   // GBK_TO_UNICODE[39568] := 16#F0A9;
   // GBK_TO_UNICODE[39569] := 16#7693;
   // GBK_TO_UNICODE[39570] := 16#F0AA;
   // GBK_TO_UNICODE[39571] := 16#7699;
   // GBK_TO_UNICODE[39572] := 16#F0AB;
   // GBK_TO_UNICODE[39573] := 16#76A4;
   // GBK_TO_UNICODE[39574] := 16#F0AC;
   // GBK_TO_UNICODE[39575] := 16#74DE;
   // GBK_TO_UNICODE[39576] := 16#F0AD;
   // GBK_TO_UNICODE[39577] := 16#74E0;
   // GBK_TO_UNICODE[39578] := 16#F0AE;
   // GBK_TO_UNICODE[39579] := 16#752C;
   // GBK_TO_UNICODE[39580] := 16#F0AF;
   // GBK_TO_UNICODE[39581] := 16#9E20;
   // GBK_TO_UNICODE[39582] := 16#F0B0;
   // GBK_TO_UNICODE[39583] := 16#9E22;
   // GBK_TO_UNICODE[39584] := 16#F0B1;
   // GBK_TO_UNICODE[39585] := 16#9E28;
   // GBK_TO_UNICODE[39586] := 16#F0B2;
   // GBK_TO_UNICODE[39587] := 16#9E29;
   // GBK_TO_UNICODE[39588] := 16#F0B3;
   // GBK_TO_UNICODE[39589] := 16#9E2A;
   // GBK_TO_UNICODE[39590] := 16#F0B4;
   // GBK_TO_UNICODE[39591] := 16#9E2B;
   // GBK_TO_UNICODE[39592] := 16#F0B5;
   // GBK_TO_UNICODE[39593] := 16#9E2C;
   // GBK_TO_UNICODE[39594] := 16#F0B6;
   // GBK_TO_UNICODE[39595] := 16#9E32;
   // GBK_TO_UNICODE[39596] := 16#F0B7;
   // GBK_TO_UNICODE[39597] := 16#9E31;
   // GBK_TO_UNICODE[39598] := 16#F0B8;
   // GBK_TO_UNICODE[39599] := 16#9E36;
   // GBK_TO_UNICODE[39600] := 16#F0B9;
   // GBK_TO_UNICODE[39601] := 16#9E38;
   // GBK_TO_UNICODE[39602] := 16#F0BA;
   // GBK_TO_UNICODE[39603] := 16#9E37;
   // GBK_TO_UNICODE[39604] := 16#F0BB;
   // GBK_TO_UNICODE[39605] := 16#9E39;
   // GBK_TO_UNICODE[39606] := 16#F0BC;
   // GBK_TO_UNICODE[39607] := 16#9E3A;
   // GBK_TO_UNICODE[39608] := 16#F0BD;
   // GBK_TO_UNICODE[39609] := 16#9E3E;
   // GBK_TO_UNICODE[39610] := 16#F0BE;
   // GBK_TO_UNICODE[39611] := 16#9E41;
   // GBK_TO_UNICODE[39612] := 16#F0BF;
   // GBK_TO_UNICODE[39613] := 16#9E42;
   // GBK_TO_UNICODE[39614] := 16#F0C0;
   // GBK_TO_UNICODE[39615] := 16#9E44;
   // GBK_TO_UNICODE[39616] := 16#F0C1;
   // GBK_TO_UNICODE[39617] := 16#9E46;
   // GBK_TO_UNICODE[39618] := 16#F0C2;
   // GBK_TO_UNICODE[39619] := 16#9E47;
   // GBK_TO_UNICODE[39620] := 16#F0C3;
   // GBK_TO_UNICODE[39621] := 16#9E48;
   // GBK_TO_UNICODE[39622] := 16#F0C4;
   // GBK_TO_UNICODE[39623] := 16#9E49;
   // GBK_TO_UNICODE[39624] := 16#F0C5;
   // GBK_TO_UNICODE[39625] := 16#9E4B;
   // GBK_TO_UNICODE[39626] := 16#F0C6;
   // GBK_TO_UNICODE[39627] := 16#9E4C;
   // GBK_TO_UNICODE[39628] := 16#F0C7;
   // GBK_TO_UNICODE[39629] := 16#9E4E;
   // GBK_TO_UNICODE[39630] := 16#F0C8;
   // GBK_TO_UNICODE[39631] := 16#9E51;
   // GBK_TO_UNICODE[39632] := 16#F0C9;
   // GBK_TO_UNICODE[39633] := 16#9E55;
   // GBK_TO_UNICODE[39634] := 16#F0CA;
   // GBK_TO_UNICODE[39635] := 16#9E57;
   // GBK_TO_UNICODE[39636] := 16#F0CB;
   // GBK_TO_UNICODE[39637] := 16#9E5A;
   // GBK_TO_UNICODE[39638] := 16#F0CC;
   // GBK_TO_UNICODE[39639] := 16#9E5B;
   // GBK_TO_UNICODE[39640] := 16#F0CD;
   // GBK_TO_UNICODE[39641] := 16#9E5C;
   // GBK_TO_UNICODE[39642] := 16#F0CE;
   // GBK_TO_UNICODE[39643] := 16#9E5E;
   // GBK_TO_UNICODE[39644] := 16#F0CF;
   // GBK_TO_UNICODE[39645] := 16#9E63;
   // GBK_TO_UNICODE[39646] := 16#F0D0;
   // GBK_TO_UNICODE[39647] := 16#9E66;
   // GBK_TO_UNICODE[39648] := 16#F0D1;
   // GBK_TO_UNICODE[39649] := 16#9E67;
   // GBK_TO_UNICODE[39650] := 16#F0D2;
   // GBK_TO_UNICODE[39651] := 16#9E68;
   // GBK_TO_UNICODE[39652] := 16#F0D3;
   // GBK_TO_UNICODE[39653] := 16#9E69;
   // GBK_TO_UNICODE[39654] := 16#F0D4;
   // GBK_TO_UNICODE[39655] := 16#9E6A;
   // GBK_TO_UNICODE[39656] := 16#F0D5;
   // GBK_TO_UNICODE[39657] := 16#9E6B;
   // GBK_TO_UNICODE[39658] := 16#F0D6;
   // GBK_TO_UNICODE[39659] := 16#9E6C;
   // GBK_TO_UNICODE[39660] := 16#F0D7;
   // GBK_TO_UNICODE[39661] := 16#9E71;
   // GBK_TO_UNICODE[39662] := 16#F0D8;
   // GBK_TO_UNICODE[39663] := 16#9E6D;
   // GBK_TO_UNICODE[39664] := 16#F0D9;
   // GBK_TO_UNICODE[39665] := 16#9E73;
   // GBK_TO_UNICODE[39666] := 16#F0DA;
   // GBK_TO_UNICODE[39667] := 16#7592;
   // GBK_TO_UNICODE[39668] := 16#F0DB;
   // GBK_TO_UNICODE[39669] := 16#7594;
   // GBK_TO_UNICODE[39670] := 16#F0DC;
   // GBK_TO_UNICODE[39671] := 16#7596;
   // GBK_TO_UNICODE[39672] := 16#F0DD;
   // GBK_TO_UNICODE[39673] := 16#75A0;
   // GBK_TO_UNICODE[39674] := 16#F0DE;
   // GBK_TO_UNICODE[39675] := 16#759D;
   // GBK_TO_UNICODE[39676] := 16#F0DF;
   // GBK_TO_UNICODE[39677] := 16#75AC;
   // GBK_TO_UNICODE[39678] := 16#F0E0;
   // GBK_TO_UNICODE[39679] := 16#75A3;
   // GBK_TO_UNICODE[39680] := 16#F0E1;
   // GBK_TO_UNICODE[39681] := 16#75B3;
   // GBK_TO_UNICODE[39682] := 16#F0E2;
   // GBK_TO_UNICODE[39683] := 16#75B4;
   // GBK_TO_UNICODE[39684] := 16#F0E3;
   // GBK_TO_UNICODE[39685] := 16#75B8;
   // GBK_TO_UNICODE[39686] := 16#F0E4;
   // GBK_TO_UNICODE[39687] := 16#75C4;
   // GBK_TO_UNICODE[39688] := 16#F0E5;
   // GBK_TO_UNICODE[39689] := 16#75B1;
   // GBK_TO_UNICODE[39690] := 16#F0E6;
   // GBK_TO_UNICODE[39691] := 16#75B0;
   // GBK_TO_UNICODE[39692] := 16#F0E7;
   // GBK_TO_UNICODE[39693] := 16#75C3;
   // GBK_TO_UNICODE[39694] := 16#F0E8;
   // GBK_TO_UNICODE[39695] := 16#75C2;
   // GBK_TO_UNICODE[39696] := 16#F0E9;
   // GBK_TO_UNICODE[39697] := 16#75D6;
   // GBK_TO_UNICODE[39698] := 16#F0EA;
   // GBK_TO_UNICODE[39699] := 16#75CD;
   // GBK_TO_UNICODE[39700] := 16#F0EB;
   // GBK_TO_UNICODE[39701] := 16#75E3;
   // GBK_TO_UNICODE[39702] := 16#F0EC;
   // GBK_TO_UNICODE[39703] := 16#75E8;
   // GBK_TO_UNICODE[39704] := 16#F0ED;
   // GBK_TO_UNICODE[39705] := 16#75E6;
   // GBK_TO_UNICODE[39706] := 16#F0EE;
   // GBK_TO_UNICODE[39707] := 16#75E4;
   // GBK_TO_UNICODE[39708] := 16#F0EF;
   // GBK_TO_UNICODE[39709] := 16#75EB;
   // GBK_TO_UNICODE[39710] := 16#F0F0;
   // GBK_TO_UNICODE[39711] := 16#75E7;
   // GBK_TO_UNICODE[39712] := 16#F0F1;
   // GBK_TO_UNICODE[39713] := 16#7603;
   // GBK_TO_UNICODE[39714] := 16#F0F2;
   // GBK_TO_UNICODE[39715] := 16#75F1;
   // GBK_TO_UNICODE[39716] := 16#F0F3;
   // GBK_TO_UNICODE[39717] := 16#75FC;
   // GBK_TO_UNICODE[39718] := 16#F0F4;
   // GBK_TO_UNICODE[39719] := 16#75FF;
   // GBK_TO_UNICODE[39720] := 16#F0F5;
   // GBK_TO_UNICODE[39721] := 16#7610;
   // GBK_TO_UNICODE[39722] := 16#F0F6;
   // GBK_TO_UNICODE[39723] := 16#7600;
   // GBK_TO_UNICODE[39724] := 16#F0F7;
   // GBK_TO_UNICODE[39725] := 16#7605;
   // GBK_TO_UNICODE[39726] := 16#F0F8;
   // GBK_TO_UNICODE[39727] := 16#760C;
   // GBK_TO_UNICODE[39728] := 16#F0F9;
   // GBK_TO_UNICODE[39729] := 16#7617;
   // GBK_TO_UNICODE[39730] := 16#F0FA;
   // GBK_TO_UNICODE[39731] := 16#760A;
   // GBK_TO_UNICODE[39732] := 16#F0FB;
   // GBK_TO_UNICODE[39733] := 16#7625;
   // GBK_TO_UNICODE[39734] := 16#F0FC;
   // GBK_TO_UNICODE[39735] := 16#7618;
   // GBK_TO_UNICODE[39736] := 16#F0FD;
   // GBK_TO_UNICODE[39737] := 16#7615;
   // GBK_TO_UNICODE[39738] := 16#F0FE;
   // GBK_TO_UNICODE[39739] := 16#7619;
   // GBK_TO_UNICODE[39740] := 16#F140;
   // GBK_TO_UNICODE[39741] := 16#998C;
   // GBK_TO_UNICODE[39742] := 16#F141;
   // GBK_TO_UNICODE[39743] := 16#998E;
   // GBK_TO_UNICODE[39744] := 16#F142;
   // GBK_TO_UNICODE[39745] := 16#999A;
   // GBK_TO_UNICODE[39746] := 16#F143;
   // GBK_TO_UNICODE[39747] := 16#999B;
   // GBK_TO_UNICODE[39748] := 16#F144;
   // GBK_TO_UNICODE[39749] := 16#999C;
   // GBK_TO_UNICODE[39750] := 16#F145;
   // GBK_TO_UNICODE[39751] := 16#999D;
   // GBK_TO_UNICODE[39752] := 16#F146;
   // GBK_TO_UNICODE[39753] := 16#999E;
   // GBK_TO_UNICODE[39754] := 16#F147;
   // GBK_TO_UNICODE[39755] := 16#999F;
   // GBK_TO_UNICODE[39756] := 16#F148;
   // GBK_TO_UNICODE[39757] := 16#99A0;
   // GBK_TO_UNICODE[39758] := 16#F149;
   // GBK_TO_UNICODE[39759] := 16#99A1;
   // GBK_TO_UNICODE[39760] := 16#F14A;
   // GBK_TO_UNICODE[39761] := 16#99A2;
   // GBK_TO_UNICODE[39762] := 16#F14B;
   // GBK_TO_UNICODE[39763] := 16#99A3;
   // GBK_TO_UNICODE[39764] := 16#F14C;
   // GBK_TO_UNICODE[39765] := 16#99A4;
   // GBK_TO_UNICODE[39766] := 16#F14D;
   // GBK_TO_UNICODE[39767] := 16#99A6;
   // GBK_TO_UNICODE[39768] := 16#F14E;
   // GBK_TO_UNICODE[39769] := 16#99A7;
   // GBK_TO_UNICODE[39770] := 16#F14F;
   // GBK_TO_UNICODE[39771] := 16#99A9;
   // GBK_TO_UNICODE[39772] := 16#F150;
   // GBK_TO_UNICODE[39773] := 16#99AA;
   // GBK_TO_UNICODE[39774] := 16#F151;
   // GBK_TO_UNICODE[39775] := 16#99AB;
   // GBK_TO_UNICODE[39776] := 16#F152;
   // GBK_TO_UNICODE[39777] := 16#99AC;
   // GBK_TO_UNICODE[39778] := 16#F153;
   // GBK_TO_UNICODE[39779] := 16#99AD;
   // GBK_TO_UNICODE[39780] := 16#F154;
   // GBK_TO_UNICODE[39781] := 16#99AE;
   // GBK_TO_UNICODE[39782] := 16#F155;
   // GBK_TO_UNICODE[39783] := 16#99AF;
   // GBK_TO_UNICODE[39784] := 16#F156;
   // GBK_TO_UNICODE[39785] := 16#99B0;
   // GBK_TO_UNICODE[39786] := 16#F157;
   // GBK_TO_UNICODE[39787] := 16#99B1;
   // GBK_TO_UNICODE[39788] := 16#F158;
   // GBK_TO_UNICODE[39789] := 16#99B2;
   // GBK_TO_UNICODE[39790] := 16#F159;
   // GBK_TO_UNICODE[39791] := 16#99B3;
   // GBK_TO_UNICODE[39792] := 16#F15A;
   // GBK_TO_UNICODE[39793] := 16#99B4;
   // GBK_TO_UNICODE[39794] := 16#F15B;
   // GBK_TO_UNICODE[39795] := 16#99B5;
   // GBK_TO_UNICODE[39796] := 16#F15C;
   // GBK_TO_UNICODE[39797] := 16#99B6;
   // GBK_TO_UNICODE[39798] := 16#F15D;
   // GBK_TO_UNICODE[39799] := 16#99B7;
   // GBK_TO_UNICODE[39800] := 16#F15E;
   // GBK_TO_UNICODE[39801] := 16#99B8;
   // GBK_TO_UNICODE[39802] := 16#F15F;
   // GBK_TO_UNICODE[39803] := 16#99B9;
   // GBK_TO_UNICODE[39804] := 16#F160;
   // GBK_TO_UNICODE[39805] := 16#99BA;
   // GBK_TO_UNICODE[39806] := 16#F161;
   // GBK_TO_UNICODE[39807] := 16#99BB;
   // GBK_TO_UNICODE[39808] := 16#F162;
   // GBK_TO_UNICODE[39809] := 16#99BC;
   // GBK_TO_UNICODE[39810] := 16#F163;
   // GBK_TO_UNICODE[39811] := 16#99BD;
   // GBK_TO_UNICODE[39812] := 16#F164;
   // GBK_TO_UNICODE[39813] := 16#99BE;
   // GBK_TO_UNICODE[39814] := 16#F165;
   // GBK_TO_UNICODE[39815] := 16#99BF;
   // GBK_TO_UNICODE[39816] := 16#F166;
   // GBK_TO_UNICODE[39817] := 16#99C0;
   // GBK_TO_UNICODE[39818] := 16#F167;
   // GBK_TO_UNICODE[39819] := 16#99C1;
   // GBK_TO_UNICODE[39820] := 16#F168;
   // GBK_TO_UNICODE[39821] := 16#99C2;
   // GBK_TO_UNICODE[39822] := 16#F169;
   // GBK_TO_UNICODE[39823] := 16#99C3;
   // GBK_TO_UNICODE[39824] := 16#F16A;
   // GBK_TO_UNICODE[39825] := 16#99C4;
   // GBK_TO_UNICODE[39826] := 16#F16B;
   // GBK_TO_UNICODE[39827] := 16#99C5;
   // GBK_TO_UNICODE[39828] := 16#F16C;
   // GBK_TO_UNICODE[39829] := 16#99C6;
   // GBK_TO_UNICODE[39830] := 16#F16D;
   // GBK_TO_UNICODE[39831] := 16#99C7;
   // GBK_TO_UNICODE[39832] := 16#F16E;
   // GBK_TO_UNICODE[39833] := 16#99C8;
   // GBK_TO_UNICODE[39834] := 16#F16F;
   // GBK_TO_UNICODE[39835] := 16#99C9;
   // GBK_TO_UNICODE[39836] := 16#F170;
   // GBK_TO_UNICODE[39837] := 16#99CA;
   // GBK_TO_UNICODE[39838] := 16#F171;
   // GBK_TO_UNICODE[39839] := 16#99CB;
   // GBK_TO_UNICODE[39840] := 16#F172;
   // GBK_TO_UNICODE[39841] := 16#99CC;
   // GBK_TO_UNICODE[39842] := 16#F173;
   // GBK_TO_UNICODE[39843] := 16#99CD;
   // GBK_TO_UNICODE[39844] := 16#F174;
   // GBK_TO_UNICODE[39845] := 16#99CE;
   // GBK_TO_UNICODE[39846] := 16#F175;
   // GBK_TO_UNICODE[39847] := 16#99CF;
   // GBK_TO_UNICODE[39848] := 16#F176;
   // GBK_TO_UNICODE[39849] := 16#99D0;
   // GBK_TO_UNICODE[39850] := 16#F177;
   // GBK_TO_UNICODE[39851] := 16#99D1;
   // GBK_TO_UNICODE[39852] := 16#F178;
   // GBK_TO_UNICODE[39853] := 16#99D2;
   // GBK_TO_UNICODE[39854] := 16#F179;
   // GBK_TO_UNICODE[39855] := 16#99D3;
   // GBK_TO_UNICODE[39856] := 16#F17A;
   // GBK_TO_UNICODE[39857] := 16#99D4;
   // GBK_TO_UNICODE[39858] := 16#F17B;
   // GBK_TO_UNICODE[39859] := 16#99D5;
   // GBK_TO_UNICODE[39860] := 16#F17C;
   // GBK_TO_UNICODE[39861] := 16#99D6;
   // GBK_TO_UNICODE[39862] := 16#F17D;
   // GBK_TO_UNICODE[39863] := 16#99D7;
   // GBK_TO_UNICODE[39864] := 16#F17E;
   // GBK_TO_UNICODE[39865] := 16#99D8;
   // GBK_TO_UNICODE[39866] := 16#F180;
   // GBK_TO_UNICODE[39867] := 16#99D9;
   // GBK_TO_UNICODE[39868] := 16#F181;
   // GBK_TO_UNICODE[39869] := 16#99DA;
   // GBK_TO_UNICODE[39870] := 16#F182;
   // GBK_TO_UNICODE[39871] := 16#99DB;
   // GBK_TO_UNICODE[39872] := 16#F183;
   // GBK_TO_UNICODE[39873] := 16#99DC;
   // GBK_TO_UNICODE[39874] := 16#F184;
   // GBK_TO_UNICODE[39875] := 16#99DD;
   // GBK_TO_UNICODE[39876] := 16#F185;
   // GBK_TO_UNICODE[39877] := 16#99DE;
   // GBK_TO_UNICODE[39878] := 16#F186;
   // GBK_TO_UNICODE[39879] := 16#99DF;
   // GBK_TO_UNICODE[39880] := 16#F187;
   // GBK_TO_UNICODE[39881] := 16#99E0;
   // GBK_TO_UNICODE[39882] := 16#F188;
   // GBK_TO_UNICODE[39883] := 16#99E1;
   // GBK_TO_UNICODE[39884] := 16#F189;
   // GBK_TO_UNICODE[39885] := 16#99E2;
   // GBK_TO_UNICODE[39886] := 16#F18A;
   // GBK_TO_UNICODE[39887] := 16#99E3;
   // GBK_TO_UNICODE[39888] := 16#F18B;
   // GBK_TO_UNICODE[39889] := 16#99E4;
   // GBK_TO_UNICODE[39890] := 16#F18C;
   // GBK_TO_UNICODE[39891] := 16#99E5;
   // GBK_TO_UNICODE[39892] := 16#F18D;
   // GBK_TO_UNICODE[39893] := 16#99E6;
   // GBK_TO_UNICODE[39894] := 16#F18E;
   // GBK_TO_UNICODE[39895] := 16#99E7;
   // GBK_TO_UNICODE[39896] := 16#F18F;
   // GBK_TO_UNICODE[39897] := 16#99E8;
   // GBK_TO_UNICODE[39898] := 16#F190;
   // GBK_TO_UNICODE[39899] := 16#99E9;
   // GBK_TO_UNICODE[39900] := 16#F191;
   // GBK_TO_UNICODE[39901] := 16#99EA;
   // GBK_TO_UNICODE[39902] := 16#F192;
   // GBK_TO_UNICODE[39903] := 16#99EB;
   // GBK_TO_UNICODE[39904] := 16#F193;
   // GBK_TO_UNICODE[39905] := 16#99EC;
   // GBK_TO_UNICODE[39906] := 16#F194;
   // GBK_TO_UNICODE[39907] := 16#99ED;
   // GBK_TO_UNICODE[39908] := 16#F195;
   // GBK_TO_UNICODE[39909] := 16#99EE;
   // GBK_TO_UNICODE[39910] := 16#F196;
   // GBK_TO_UNICODE[39911] := 16#99EF;
   // GBK_TO_UNICODE[39912] := 16#F197;
   // GBK_TO_UNICODE[39913] := 16#99F0;
   // GBK_TO_UNICODE[39914] := 16#F198;
   // GBK_TO_UNICODE[39915] := 16#99F1;
   // GBK_TO_UNICODE[39916] := 16#F199;
   // GBK_TO_UNICODE[39917] := 16#99F2;
   // GBK_TO_UNICODE[39918] := 16#F19A;
   // GBK_TO_UNICODE[39919] := 16#99F3;
   // GBK_TO_UNICODE[39920] := 16#F19B;
   // GBK_TO_UNICODE[39921] := 16#99F4;
   // GBK_TO_UNICODE[39922] := 16#F19C;
   // GBK_TO_UNICODE[39923] := 16#99F5;
   // GBK_TO_UNICODE[39924] := 16#F19D;
   // GBK_TO_UNICODE[39925] := 16#99F6;
   // GBK_TO_UNICODE[39926] := 16#F19E;
   // GBK_TO_UNICODE[39927] := 16#99F7;
   // GBK_TO_UNICODE[39928] := 16#F19F;
   // GBK_TO_UNICODE[39929] := 16#99F8;
   // GBK_TO_UNICODE[39930] := 16#F1A0;
   // GBK_TO_UNICODE[39931] := 16#99F9;
   // GBK_TO_UNICODE[39932] := 16#F1A1;
   // GBK_TO_UNICODE[39933] := 16#761B;
   // GBK_TO_UNICODE[39934] := 16#F1A2;
   // GBK_TO_UNICODE[39935] := 16#763C;
   // GBK_TO_UNICODE[39936] := 16#F1A3;
   // GBK_TO_UNICODE[39937] := 16#7622;
   // GBK_TO_UNICODE[39938] := 16#F1A4;
   // GBK_TO_UNICODE[39939] := 16#7620;
   // GBK_TO_UNICODE[39940] := 16#F1A5;
   // GBK_TO_UNICODE[39941] := 16#7640;
   // GBK_TO_UNICODE[39942] := 16#F1A6;
   // GBK_TO_UNICODE[39943] := 16#762D;
   // GBK_TO_UNICODE[39944] := 16#F1A7;
   // GBK_TO_UNICODE[39945] := 16#7630;
   // GBK_TO_UNICODE[39946] := 16#F1A8;
   // GBK_TO_UNICODE[39947] := 16#763F;
   // GBK_TO_UNICODE[39948] := 16#F1A9;
   // GBK_TO_UNICODE[39949] := 16#7635;
   // GBK_TO_UNICODE[39950] := 16#F1AA;
   // GBK_TO_UNICODE[39951] := 16#7643;
   // GBK_TO_UNICODE[39952] := 16#F1AB;
   // GBK_TO_UNICODE[39953] := 16#763E;
   // GBK_TO_UNICODE[39954] := 16#F1AC;
   // GBK_TO_UNICODE[39955] := 16#7633;
   // GBK_TO_UNICODE[39956] := 16#F1AD;
   // GBK_TO_UNICODE[39957] := 16#764D;
   // GBK_TO_UNICODE[39958] := 16#F1AE;
   // GBK_TO_UNICODE[39959] := 16#765E;
   // GBK_TO_UNICODE[39960] := 16#F1AF;
   // GBK_TO_UNICODE[39961] := 16#7654;
   // GBK_TO_UNICODE[39962] := 16#F1B0;
   // GBK_TO_UNICODE[39963] := 16#765C;
   // GBK_TO_UNICODE[39964] := 16#F1B1;
   // GBK_TO_UNICODE[39965] := 16#7656;
   // GBK_TO_UNICODE[39966] := 16#F1B2;
   // GBK_TO_UNICODE[39967] := 16#766B;
   // GBK_TO_UNICODE[39968] := 16#F1B3;
   // GBK_TO_UNICODE[39969] := 16#766F;
   // GBK_TO_UNICODE[39970] := 16#F1B4;
   // GBK_TO_UNICODE[39971] := 16#7FCA;
   // GBK_TO_UNICODE[39972] := 16#F1B5;
   // GBK_TO_UNICODE[39973] := 16#7AE6;
   // GBK_TO_UNICODE[39974] := 16#F1B6;
   // GBK_TO_UNICODE[39975] := 16#7A78;
   // GBK_TO_UNICODE[39976] := 16#F1B7;
   // GBK_TO_UNICODE[39977] := 16#7A79;
   // GBK_TO_UNICODE[39978] := 16#F1B8;
   // GBK_TO_UNICODE[39979] := 16#7A80;
   // GBK_TO_UNICODE[39980] := 16#F1B9;
   // GBK_TO_UNICODE[39981] := 16#7A86;
   // GBK_TO_UNICODE[39982] := 16#F1BA;
   // GBK_TO_UNICODE[39983] := 16#7A88;
   // GBK_TO_UNICODE[39984] := 16#F1BB;
   // GBK_TO_UNICODE[39985] := 16#7A95;
   // GBK_TO_UNICODE[39986] := 16#F1BC;
   // GBK_TO_UNICODE[39987] := 16#7AA6;
   // GBK_TO_UNICODE[39988] := 16#F1BD;
   // GBK_TO_UNICODE[39989] := 16#7AA0;
   // GBK_TO_UNICODE[39990] := 16#F1BE;
   // GBK_TO_UNICODE[39991] := 16#7AAC;
   // GBK_TO_UNICODE[39992] := 16#F1BF;
   // GBK_TO_UNICODE[39993] := 16#7AA8;
   // GBK_TO_UNICODE[39994] := 16#F1C0;
   // GBK_TO_UNICODE[39995] := 16#7AAD;
   // GBK_TO_UNICODE[39996] := 16#F1C1;
   // GBK_TO_UNICODE[39997] := 16#7AB3;
   // GBK_TO_UNICODE[39998] := 16#F1C2;
   // GBK_TO_UNICODE[39999] := 16#8864;
   // GBK_TO_UNICODE[40000] := 16#F1C3;
   // GBK_TO_UNICODE[40001] := 16#8869;
   // GBK_TO_UNICODE[40002] := 16#F1C4;
   // GBK_TO_UNICODE[40003] := 16#8872;
   // GBK_TO_UNICODE[40004] := 16#F1C5;
   // GBK_TO_UNICODE[40005] := 16#887D;
   // GBK_TO_UNICODE[40006] := 16#F1C6;
   // GBK_TO_UNICODE[40007] := 16#887F;
   // GBK_TO_UNICODE[40008] := 16#F1C7;
   // GBK_TO_UNICODE[40009] := 16#8882;
   // GBK_TO_UNICODE[40010] := 16#F1C8;
   // GBK_TO_UNICODE[40011] := 16#88A2;
   // GBK_TO_UNICODE[40012] := 16#F1C9;
   // GBK_TO_UNICODE[40013] := 16#88C6;
   // GBK_TO_UNICODE[40014] := 16#F1CA;
   // GBK_TO_UNICODE[40015] := 16#88B7;
   // GBK_TO_UNICODE[40016] := 16#F1CB;
   // GBK_TO_UNICODE[40017] := 16#88BC;
   // GBK_TO_UNICODE[40018] := 16#F1CC;
   // GBK_TO_UNICODE[40019] := 16#88C9;
   // GBK_TO_UNICODE[40020] := 16#F1CD;
   // GBK_TO_UNICODE[40021] := 16#88E2;
   // GBK_TO_UNICODE[40022] := 16#F1CE;
   // GBK_TO_UNICODE[40023] := 16#88CE;
   // GBK_TO_UNICODE[40024] := 16#F1CF;
   // GBK_TO_UNICODE[40025] := 16#88E3;
   // GBK_TO_UNICODE[40026] := 16#F1D0;
   // GBK_TO_UNICODE[40027] := 16#88E5;
   // GBK_TO_UNICODE[40028] := 16#F1D1;
   // GBK_TO_UNICODE[40029] := 16#88F1;
   // GBK_TO_UNICODE[40030] := 16#F1D2;
   // GBK_TO_UNICODE[40031] := 16#891A;
   // GBK_TO_UNICODE[40032] := 16#F1D3;
   // GBK_TO_UNICODE[40033] := 16#88FC;
   // GBK_TO_UNICODE[40034] := 16#F1D4;
   // GBK_TO_UNICODE[40035] := 16#88E8;
   // GBK_TO_UNICODE[40036] := 16#F1D5;
   // GBK_TO_UNICODE[40037] := 16#88FE;
   // GBK_TO_UNICODE[40038] := 16#F1D6;
   // GBK_TO_UNICODE[40039] := 16#88F0;
   // GBK_TO_UNICODE[40040] := 16#F1D7;
   // GBK_TO_UNICODE[40041] := 16#8921;
   // GBK_TO_UNICODE[40042] := 16#F1D8;
   // GBK_TO_UNICODE[40043] := 16#8919;
   // GBK_TO_UNICODE[40044] := 16#F1D9;
   // GBK_TO_UNICODE[40045] := 16#8913;
   // GBK_TO_UNICODE[40046] := 16#F1DA;
   // GBK_TO_UNICODE[40047] := 16#891B;
   // GBK_TO_UNICODE[40048] := 16#F1DB;
   // GBK_TO_UNICODE[40049] := 16#890A;
   // GBK_TO_UNICODE[40050] := 16#F1DC;
   // GBK_TO_UNICODE[40051] := 16#8934;
   // GBK_TO_UNICODE[40052] := 16#F1DD;
   // GBK_TO_UNICODE[40053] := 16#892B;
   // GBK_TO_UNICODE[40054] := 16#F1DE;
   // GBK_TO_UNICODE[40055] := 16#8936;
   // GBK_TO_UNICODE[40056] := 16#F1DF;
   // GBK_TO_UNICODE[40057] := 16#8941;
   // GBK_TO_UNICODE[40058] := 16#F1E0;
   // GBK_TO_UNICODE[40059] := 16#8966;
   // GBK_TO_UNICODE[40060] := 16#F1E1;
   // GBK_TO_UNICODE[40061] := 16#897B;
   // GBK_TO_UNICODE[40062] := 16#F1E2;
   // GBK_TO_UNICODE[40063] := 16#758B;
   // GBK_TO_UNICODE[40064] := 16#F1E3;
   // GBK_TO_UNICODE[40065] := 16#80E5;
   // GBK_TO_UNICODE[40066] := 16#F1E4;
   // GBK_TO_UNICODE[40067] := 16#76B2;
   // GBK_TO_UNICODE[40068] := 16#F1E5;
   // GBK_TO_UNICODE[40069] := 16#76B4;
   // GBK_TO_UNICODE[40070] := 16#F1E6;
   // GBK_TO_UNICODE[40071] := 16#77DC;
   // GBK_TO_UNICODE[40072] := 16#F1E7;
   // GBK_TO_UNICODE[40073] := 16#8012;
   // GBK_TO_UNICODE[40074] := 16#F1E8;
   // GBK_TO_UNICODE[40075] := 16#8014;
   // GBK_TO_UNICODE[40076] := 16#F1E9;
   // GBK_TO_UNICODE[40077] := 16#8016;
   // GBK_TO_UNICODE[40078] := 16#F1EA;
   // GBK_TO_UNICODE[40079] := 16#801C;
   // GBK_TO_UNICODE[40080] := 16#F1EB;
   // GBK_TO_UNICODE[40081] := 16#8020;
   // GBK_TO_UNICODE[40082] := 16#F1EC;
   // GBK_TO_UNICODE[40083] := 16#8022;
   // GBK_TO_UNICODE[40084] := 16#F1ED;
   // GBK_TO_UNICODE[40085] := 16#8025;
   // GBK_TO_UNICODE[40086] := 16#F1EE;
   // GBK_TO_UNICODE[40087] := 16#8026;
   // GBK_TO_UNICODE[40088] := 16#F1EF;
   // GBK_TO_UNICODE[40089] := 16#8027;
   // GBK_TO_UNICODE[40090] := 16#F1F0;
   // GBK_TO_UNICODE[40091] := 16#8029;
   // GBK_TO_UNICODE[40092] := 16#F1F1;
   // GBK_TO_UNICODE[40093] := 16#8028;
   // GBK_TO_UNICODE[40094] := 16#F1F2;
   // GBK_TO_UNICODE[40095] := 16#8031;
   // GBK_TO_UNICODE[40096] := 16#F1F3;
   // GBK_TO_UNICODE[40097] := 16#800B;
   // GBK_TO_UNICODE[40098] := 16#F1F4;
   // GBK_TO_UNICODE[40099] := 16#8035;
   // GBK_TO_UNICODE[40100] := 16#F1F5;
   // GBK_TO_UNICODE[40101] := 16#8043;
   // GBK_TO_UNICODE[40102] := 16#F1F6;
   // GBK_TO_UNICODE[40103] := 16#8046;
   // GBK_TO_UNICODE[40104] := 16#F1F7;
   // GBK_TO_UNICODE[40105] := 16#804D;
   // GBK_TO_UNICODE[40106] := 16#F1F8;
   // GBK_TO_UNICODE[40107] := 16#8052;
   // GBK_TO_UNICODE[40108] := 16#F1F9;
   // GBK_TO_UNICODE[40109] := 16#8069;
   // GBK_TO_UNICODE[40110] := 16#F1FA;
   // GBK_TO_UNICODE[40111] := 16#8071;
   // GBK_TO_UNICODE[40112] := 16#F1FB;
   // GBK_TO_UNICODE[40113] := 16#8983;
   // GBK_TO_UNICODE[40114] := 16#F1FC;
   // GBK_TO_UNICODE[40115] := 16#9878;
   // GBK_TO_UNICODE[40116] := 16#F1FD;
   // GBK_TO_UNICODE[40117] := 16#9880;
   // GBK_TO_UNICODE[40118] := 16#F1FE;
   // GBK_TO_UNICODE[40119] := 16#9883;
   // GBK_TO_UNICODE[40120] := 16#F240;
   // GBK_TO_UNICODE[40121] := 16#99FA;
   // GBK_TO_UNICODE[40122] := 16#F241;
   // GBK_TO_UNICODE[40123] := 16#99FB;
   // GBK_TO_UNICODE[40124] := 16#F242;
   // GBK_TO_UNICODE[40125] := 16#99FC;
   // GBK_TO_UNICODE[40126] := 16#F243;
   // GBK_TO_UNICODE[40127] := 16#99FD;
   // GBK_TO_UNICODE[40128] := 16#F244;
   // GBK_TO_UNICODE[40129] := 16#99FE;
   // GBK_TO_UNICODE[40130] := 16#F245;
   // GBK_TO_UNICODE[40131] := 16#99FF;
   // GBK_TO_UNICODE[40132] := 16#F246;
   // GBK_TO_UNICODE[40133] := 16#9A00;
   // GBK_TO_UNICODE[40134] := 16#F247;
   // GBK_TO_UNICODE[40135] := 16#9A01;
   // GBK_TO_UNICODE[40136] := 16#F248;
   // GBK_TO_UNICODE[40137] := 16#9A02;
   // GBK_TO_UNICODE[40138] := 16#F249;
   // GBK_TO_UNICODE[40139] := 16#9A03;
   // GBK_TO_UNICODE[40140] := 16#F24A;
   // GBK_TO_UNICODE[40141] := 16#9A04;
   // GBK_TO_UNICODE[40142] := 16#F24B;
   // GBK_TO_UNICODE[40143] := 16#9A05;
   // GBK_TO_UNICODE[40144] := 16#F24C;
   // GBK_TO_UNICODE[40145] := 16#9A06;
   // GBK_TO_UNICODE[40146] := 16#F24D;
   // GBK_TO_UNICODE[40147] := 16#9A07;
   // GBK_TO_UNICODE[40148] := 16#F24E;
   // GBK_TO_UNICODE[40149] := 16#9A08;
   // GBK_TO_UNICODE[40150] := 16#F24F;
   // GBK_TO_UNICODE[40151] := 16#9A09;
   // GBK_TO_UNICODE[40152] := 16#F250;
   // GBK_TO_UNICODE[40153] := 16#9A0A;
   // GBK_TO_UNICODE[40154] := 16#F251;
   // GBK_TO_UNICODE[40155] := 16#9A0B;
   // GBK_TO_UNICODE[40156] := 16#F252;
   // GBK_TO_UNICODE[40157] := 16#9A0C;
   // GBK_TO_UNICODE[40158] := 16#F253;
   // GBK_TO_UNICODE[40159] := 16#9A0D;
   // GBK_TO_UNICODE[40160] := 16#F254;
   // GBK_TO_UNICODE[40161] := 16#9A0E;
   // GBK_TO_UNICODE[40162] := 16#F255;
   // GBK_TO_UNICODE[40163] := 16#9A0F;
   // GBK_TO_UNICODE[40164] := 16#F256;
   // GBK_TO_UNICODE[40165] := 16#9A10;
   // GBK_TO_UNICODE[40166] := 16#F257;
   // GBK_TO_UNICODE[40167] := 16#9A11;
   // GBK_TO_UNICODE[40168] := 16#F258;
   // GBK_TO_UNICODE[40169] := 16#9A12;
   // GBK_TO_UNICODE[40170] := 16#F259;
   // GBK_TO_UNICODE[40171] := 16#9A13;
   // GBK_TO_UNICODE[40172] := 16#F25A;
   // GBK_TO_UNICODE[40173] := 16#9A14;
   // GBK_TO_UNICODE[40174] := 16#F25B;
   // GBK_TO_UNICODE[40175] := 16#9A15;
   // GBK_TO_UNICODE[40176] := 16#F25C;
   // GBK_TO_UNICODE[40177] := 16#9A16;
   // GBK_TO_UNICODE[40178] := 16#F25D;
   // GBK_TO_UNICODE[40179] := 16#9A17;
   // GBK_TO_UNICODE[40180] := 16#F25E;
   // GBK_TO_UNICODE[40181] := 16#9A18;
   // GBK_TO_UNICODE[40182] := 16#F25F;
   // GBK_TO_UNICODE[40183] := 16#9A19;
   // GBK_TO_UNICODE[40184] := 16#F260;
   // GBK_TO_UNICODE[40185] := 16#9A1A;
   // GBK_TO_UNICODE[40186] := 16#F261;
   // GBK_TO_UNICODE[40187] := 16#9A1B;
   // GBK_TO_UNICODE[40188] := 16#F262;
   // GBK_TO_UNICODE[40189] := 16#9A1C;
   // GBK_TO_UNICODE[40190] := 16#F263;
   // GBK_TO_UNICODE[40191] := 16#9A1D;
   // GBK_TO_UNICODE[40192] := 16#F264;
   // GBK_TO_UNICODE[40193] := 16#9A1E;
   // GBK_TO_UNICODE[40194] := 16#F265;
   // GBK_TO_UNICODE[40195] := 16#9A1F;
   // GBK_TO_UNICODE[40196] := 16#F266;
   // GBK_TO_UNICODE[40197] := 16#9A20;
   // GBK_TO_UNICODE[40198] := 16#F267;
   // GBK_TO_UNICODE[40199] := 16#9A21;
   // GBK_TO_UNICODE[40200] := 16#F268;
   // GBK_TO_UNICODE[40201] := 16#9A22;
   // GBK_TO_UNICODE[40202] := 16#F269;
   // GBK_TO_UNICODE[40203] := 16#9A23;
   // GBK_TO_UNICODE[40204] := 16#F26A;
   // GBK_TO_UNICODE[40205] := 16#9A24;
   // GBK_TO_UNICODE[40206] := 16#F26B;
   // GBK_TO_UNICODE[40207] := 16#9A25;
   // GBK_TO_UNICODE[40208] := 16#F26C;
   // GBK_TO_UNICODE[40209] := 16#9A26;
   // GBK_TO_UNICODE[40210] := 16#F26D;
   // GBK_TO_UNICODE[40211] := 16#9A27;
   // GBK_TO_UNICODE[40212] := 16#F26E;
   // GBK_TO_UNICODE[40213] := 16#9A28;
   // GBK_TO_UNICODE[40214] := 16#F26F;
   // GBK_TO_UNICODE[40215] := 16#9A29;
   // GBK_TO_UNICODE[40216] := 16#F270;
   // GBK_TO_UNICODE[40217] := 16#9A2A;
   // GBK_TO_UNICODE[40218] := 16#F271;
   // GBK_TO_UNICODE[40219] := 16#9A2B;
   // GBK_TO_UNICODE[40220] := 16#F272;
   // GBK_TO_UNICODE[40221] := 16#9A2C;
   // GBK_TO_UNICODE[40222] := 16#F273;
   // GBK_TO_UNICODE[40223] := 16#9A2D;
   // GBK_TO_UNICODE[40224] := 16#F274;
   // GBK_TO_UNICODE[40225] := 16#9A2E;
   // GBK_TO_UNICODE[40226] := 16#F275;
   // GBK_TO_UNICODE[40227] := 16#9A2F;
   // GBK_TO_UNICODE[40228] := 16#F276;
   // GBK_TO_UNICODE[40229] := 16#9A30;
   // GBK_TO_UNICODE[40230] := 16#F277;
   // GBK_TO_UNICODE[40231] := 16#9A31;
   // GBK_TO_UNICODE[40232] := 16#F278;
   // GBK_TO_UNICODE[40233] := 16#9A32;
   // GBK_TO_UNICODE[40234] := 16#F279;
   // GBK_TO_UNICODE[40235] := 16#9A33;
   // GBK_TO_UNICODE[40236] := 16#F27A;
   // GBK_TO_UNICODE[40237] := 16#9A34;
   // GBK_TO_UNICODE[40238] := 16#F27B;
   // GBK_TO_UNICODE[40239] := 16#9A35;
   // GBK_TO_UNICODE[40240] := 16#F27C;
   // GBK_TO_UNICODE[40241] := 16#9A36;
   // GBK_TO_UNICODE[40242] := 16#F27D;
   // GBK_TO_UNICODE[40243] := 16#9A37;
   // GBK_TO_UNICODE[40244] := 16#F27E;
   // GBK_TO_UNICODE[40245] := 16#9A38;
   // GBK_TO_UNICODE[40246] := 16#F280;
   // GBK_TO_UNICODE[40247] := 16#9A39;
   // GBK_TO_UNICODE[40248] := 16#F281;
   // GBK_TO_UNICODE[40249] := 16#9A3A;
   // GBK_TO_UNICODE[40250] := 16#F282;
   // GBK_TO_UNICODE[40251] := 16#9A3B;
   // GBK_TO_UNICODE[40252] := 16#F283;
   // GBK_TO_UNICODE[40253] := 16#9A3C;
   // GBK_TO_UNICODE[40254] := 16#F284;
   // GBK_TO_UNICODE[40255] := 16#9A3D;
   // GBK_TO_UNICODE[40256] := 16#F285;
   // GBK_TO_UNICODE[40257] := 16#9A3E;
   // GBK_TO_UNICODE[40258] := 16#F286;
   // GBK_TO_UNICODE[40259] := 16#9A3F;
   // GBK_TO_UNICODE[40260] := 16#F287;
   // GBK_TO_UNICODE[40261] := 16#9A40;
   // GBK_TO_UNICODE[40262] := 16#F288;
   // GBK_TO_UNICODE[40263] := 16#9A41;
   // GBK_TO_UNICODE[40264] := 16#F289;
   // GBK_TO_UNICODE[40265] := 16#9A42;
   // GBK_TO_UNICODE[40266] := 16#F28A;
   // GBK_TO_UNICODE[40267] := 16#9A43;
   // GBK_TO_UNICODE[40268] := 16#F28B;
   // GBK_TO_UNICODE[40269] := 16#9A44;
   // GBK_TO_UNICODE[40270] := 16#F28C;
   // GBK_TO_UNICODE[40271] := 16#9A45;
   // GBK_TO_UNICODE[40272] := 16#F28D;
   // GBK_TO_UNICODE[40273] := 16#9A46;
   // GBK_TO_UNICODE[40274] := 16#F28E;
   // GBK_TO_UNICODE[40275] := 16#9A47;
   // GBK_TO_UNICODE[40276] := 16#F28F;
   // GBK_TO_UNICODE[40277] := 16#9A48;
   // GBK_TO_UNICODE[40278] := 16#F290;
   // GBK_TO_UNICODE[40279] := 16#9A49;
   // GBK_TO_UNICODE[40280] := 16#F291;
   // GBK_TO_UNICODE[40281] := 16#9A4A;
   // GBK_TO_UNICODE[40282] := 16#F292;
   // GBK_TO_UNICODE[40283] := 16#9A4B;
   // GBK_TO_UNICODE[40284] := 16#F293;
   // GBK_TO_UNICODE[40285] := 16#9A4C;
   // GBK_TO_UNICODE[40286] := 16#F294;
   // GBK_TO_UNICODE[40287] := 16#9A4D;
   // GBK_TO_UNICODE[40288] := 16#F295;
   // GBK_TO_UNICODE[40289] := 16#9A4E;
   // GBK_TO_UNICODE[40290] := 16#F296;
   // GBK_TO_UNICODE[40291] := 16#9A4F;
   // GBK_TO_UNICODE[40292] := 16#F297;
   // GBK_TO_UNICODE[40293] := 16#9A50;
   // GBK_TO_UNICODE[40294] := 16#F298;
   // GBK_TO_UNICODE[40295] := 16#9A51;
   // GBK_TO_UNICODE[40296] := 16#F299;
   // GBK_TO_UNICODE[40297] := 16#9A52;
   // GBK_TO_UNICODE[40298] := 16#F29A;
   // GBK_TO_UNICODE[40299] := 16#9A53;
   // GBK_TO_UNICODE[40300] := 16#F29B;
   // GBK_TO_UNICODE[40301] := 16#9A54;
   // GBK_TO_UNICODE[40302] := 16#F29C;
   // GBK_TO_UNICODE[40303] := 16#9A55;
   // GBK_TO_UNICODE[40304] := 16#F29D;
   // GBK_TO_UNICODE[40305] := 16#9A56;
   // GBK_TO_UNICODE[40306] := 16#F29E;
   // GBK_TO_UNICODE[40307] := 16#9A57;
   // GBK_TO_UNICODE[40308] := 16#F29F;
   // GBK_TO_UNICODE[40309] := 16#9A58;
   // GBK_TO_UNICODE[40310] := 16#F2A0;
   // GBK_TO_UNICODE[40311] := 16#9A59;
   // GBK_TO_UNICODE[40312] := 16#F2A1;
   // GBK_TO_UNICODE[40313] := 16#9889;
   // GBK_TO_UNICODE[40314] := 16#F2A2;
   // GBK_TO_UNICODE[40315] := 16#988C;
   // GBK_TO_UNICODE[40316] := 16#F2A3;
   // GBK_TO_UNICODE[40317] := 16#988D;
   // GBK_TO_UNICODE[40318] := 16#F2A4;
   // GBK_TO_UNICODE[40319] := 16#988F;
   // GBK_TO_UNICODE[40320] := 16#F2A5;
   // GBK_TO_UNICODE[40321] := 16#9894;
   // GBK_TO_UNICODE[40322] := 16#F2A6;
   // GBK_TO_UNICODE[40323] := 16#989A;
   // GBK_TO_UNICODE[40324] := 16#F2A7;
   // GBK_TO_UNICODE[40325] := 16#989B;
   // GBK_TO_UNICODE[40326] := 16#F2A8;
   // GBK_TO_UNICODE[40327] := 16#989E;
   // GBK_TO_UNICODE[40328] := 16#F2A9;
   // GBK_TO_UNICODE[40329] := 16#989F;
   // GBK_TO_UNICODE[40330] := 16#F2AA;
   // GBK_TO_UNICODE[40331] := 16#98A1;
   // GBK_TO_UNICODE[40332] := 16#F2AB;
   // GBK_TO_UNICODE[40333] := 16#98A2;
   // GBK_TO_UNICODE[40334] := 16#F2AC;
   // GBK_TO_UNICODE[40335] := 16#98A5;
   // GBK_TO_UNICODE[40336] := 16#F2AD;
   // GBK_TO_UNICODE[40337] := 16#98A6;
   // GBK_TO_UNICODE[40338] := 16#F2AE;
   // GBK_TO_UNICODE[40339] := 16#864D;
   // GBK_TO_UNICODE[40340] := 16#F2AF;
   // GBK_TO_UNICODE[40341] := 16#8654;
   // GBK_TO_UNICODE[40342] := 16#F2B0;
   // GBK_TO_UNICODE[40343] := 16#866C;
   // GBK_TO_UNICODE[40344] := 16#F2B1;
   // GBK_TO_UNICODE[40345] := 16#866E;
   // GBK_TO_UNICODE[40346] := 16#F2B2;
   // GBK_TO_UNICODE[40347] := 16#867F;
   // GBK_TO_UNICODE[40348] := 16#F2B3;
   // GBK_TO_UNICODE[40349] := 16#867A;
   // GBK_TO_UNICODE[40350] := 16#F2B4;
   // GBK_TO_UNICODE[40351] := 16#867C;
   // GBK_TO_UNICODE[40352] := 16#F2B5;
   // GBK_TO_UNICODE[40353] := 16#867B;
   // GBK_TO_UNICODE[40354] := 16#F2B6;
   // GBK_TO_UNICODE[40355] := 16#86A8;
   // GBK_TO_UNICODE[40356] := 16#F2B7;
   // GBK_TO_UNICODE[40357] := 16#868D;
   // GBK_TO_UNICODE[40358] := 16#F2B8;
   // GBK_TO_UNICODE[40359] := 16#868B;
   // GBK_TO_UNICODE[40360] := 16#F2B9;
   // GBK_TO_UNICODE[40361] := 16#86AC;
   // GBK_TO_UNICODE[40362] := 16#F2BA;
   // GBK_TO_UNICODE[40363] := 16#869D;
   // GBK_TO_UNICODE[40364] := 16#F2BB;
   // GBK_TO_UNICODE[40365] := 16#86A7;
   // GBK_TO_UNICODE[40366] := 16#F2BC;
   // GBK_TO_UNICODE[40367] := 16#86A3;
   // GBK_TO_UNICODE[40368] := 16#F2BD;
   // GBK_TO_UNICODE[40369] := 16#86AA;
   // GBK_TO_UNICODE[40370] := 16#F2BE;
   // GBK_TO_UNICODE[40371] := 16#8693;
   // GBK_TO_UNICODE[40372] := 16#F2BF;
   // GBK_TO_UNICODE[40373] := 16#86A9;
   // GBK_TO_UNICODE[40374] := 16#F2C0;
   // GBK_TO_UNICODE[40375] := 16#86B6;
   // GBK_TO_UNICODE[40376] := 16#F2C1;
   // GBK_TO_UNICODE[40377] := 16#86C4;
   // GBK_TO_UNICODE[40378] := 16#F2C2;
   // GBK_TO_UNICODE[40379] := 16#86B5;
   // GBK_TO_UNICODE[40380] := 16#F2C3;
   // GBK_TO_UNICODE[40381] := 16#86CE;
   // GBK_TO_UNICODE[40382] := 16#F2C4;
   // GBK_TO_UNICODE[40383] := 16#86B0;
   // GBK_TO_UNICODE[40384] := 16#F2C5;
   // GBK_TO_UNICODE[40385] := 16#86BA;
   // GBK_TO_UNICODE[40386] := 16#F2C6;
   // GBK_TO_UNICODE[40387] := 16#86B1;
   // GBK_TO_UNICODE[40388] := 16#F2C7;
   // GBK_TO_UNICODE[40389] := 16#86AF;
   // GBK_TO_UNICODE[40390] := 16#F2C8;
   // GBK_TO_UNICODE[40391] := 16#86C9;
   // GBK_TO_UNICODE[40392] := 16#F2C9;
   // GBK_TO_UNICODE[40393] := 16#86CF;
   // GBK_TO_UNICODE[40394] := 16#F2CA;
   // GBK_TO_UNICODE[40395] := 16#86B4;
   // GBK_TO_UNICODE[40396] := 16#F2CB;
   // GBK_TO_UNICODE[40397] := 16#86E9;
   // GBK_TO_UNICODE[40398] := 16#F2CC;
   // GBK_TO_UNICODE[40399] := 16#86F1;
   // GBK_TO_UNICODE[40400] := 16#F2CD;
   // GBK_TO_UNICODE[40401] := 16#86F2;
   // GBK_TO_UNICODE[40402] := 16#F2CE;
   // GBK_TO_UNICODE[40403] := 16#86ED;
   // GBK_TO_UNICODE[40404] := 16#F2CF;
   // GBK_TO_UNICODE[40405] := 16#86F3;
   // GBK_TO_UNICODE[40406] := 16#F2D0;
   // GBK_TO_UNICODE[40407] := 16#86D0;
   // GBK_TO_UNICODE[40408] := 16#F2D1;
   // GBK_TO_UNICODE[40409] := 16#8713;
   // GBK_TO_UNICODE[40410] := 16#F2D2;
   // GBK_TO_UNICODE[40411] := 16#86DE;
   // GBK_TO_UNICODE[40412] := 16#F2D3;
   // GBK_TO_UNICODE[40413] := 16#86F4;
   // GBK_TO_UNICODE[40414] := 16#F2D4;
   // GBK_TO_UNICODE[40415] := 16#86DF;
   // GBK_TO_UNICODE[40416] := 16#F2D5;
   // GBK_TO_UNICODE[40417] := 16#86D8;
   // GBK_TO_UNICODE[40418] := 16#F2D6;
   // GBK_TO_UNICODE[40419] := 16#86D1;
   // GBK_TO_UNICODE[40420] := 16#F2D7;
   // GBK_TO_UNICODE[40421] := 16#8703;
   // GBK_TO_UNICODE[40422] := 16#F2D8;
   // GBK_TO_UNICODE[40423] := 16#8707;
   // GBK_TO_UNICODE[40424] := 16#F2D9;
   // GBK_TO_UNICODE[40425] := 16#86F8;
   // GBK_TO_UNICODE[40426] := 16#F2DA;
   // GBK_TO_UNICODE[40427] := 16#8708;
   // GBK_TO_UNICODE[40428] := 16#F2DB;
   // GBK_TO_UNICODE[40429] := 16#870A;
   // GBK_TO_UNICODE[40430] := 16#F2DC;
   // GBK_TO_UNICODE[40431] := 16#870D;
   // GBK_TO_UNICODE[40432] := 16#F2DD;
   // GBK_TO_UNICODE[40433] := 16#8709;
   // GBK_TO_UNICODE[40434] := 16#F2DE;
   // GBK_TO_UNICODE[40435] := 16#8723;
   // GBK_TO_UNICODE[40436] := 16#F2DF;
   // GBK_TO_UNICODE[40437] := 16#873B;
   // GBK_TO_UNICODE[40438] := 16#F2E0;
   // GBK_TO_UNICODE[40439] := 16#871E;
   // GBK_TO_UNICODE[40440] := 16#F2E1;
   // GBK_TO_UNICODE[40441] := 16#8725;
   // GBK_TO_UNICODE[40442] := 16#F2E2;
   // GBK_TO_UNICODE[40443] := 16#872E;
   // GBK_TO_UNICODE[40444] := 16#F2E3;
   // GBK_TO_UNICODE[40445] := 16#871A;
   // GBK_TO_UNICODE[40446] := 16#F2E4;
   // GBK_TO_UNICODE[40447] := 16#873E;
   // GBK_TO_UNICODE[40448] := 16#F2E5;
   // GBK_TO_UNICODE[40449] := 16#8748;
   // GBK_TO_UNICODE[40450] := 16#F2E6;
   // GBK_TO_UNICODE[40451] := 16#8734;
   // GBK_TO_UNICODE[40452] := 16#F2E7;
   // GBK_TO_UNICODE[40453] := 16#8731;
   // GBK_TO_UNICODE[40454] := 16#F2E8;
   // GBK_TO_UNICODE[40455] := 16#8729;
   // GBK_TO_UNICODE[40456] := 16#F2E9;
   // GBK_TO_UNICODE[40457] := 16#8737;
   // GBK_TO_UNICODE[40458] := 16#F2EA;
   // GBK_TO_UNICODE[40459] := 16#873F;
   // GBK_TO_UNICODE[40460] := 16#F2EB;
   // GBK_TO_UNICODE[40461] := 16#8782;
   // GBK_TO_UNICODE[40462] := 16#F2EC;
   // GBK_TO_UNICODE[40463] := 16#8722;
   // GBK_TO_UNICODE[40464] := 16#F2ED;
   // GBK_TO_UNICODE[40465] := 16#877D;
   // GBK_TO_UNICODE[40466] := 16#F2EE;
   // GBK_TO_UNICODE[40467] := 16#877E;
   // GBK_TO_UNICODE[40468] := 16#F2EF;
   // GBK_TO_UNICODE[40469] := 16#877B;
   // GBK_TO_UNICODE[40470] := 16#F2F0;
   // GBK_TO_UNICODE[40471] := 16#8760;
   // GBK_TO_UNICODE[40472] := 16#F2F1;
   // GBK_TO_UNICODE[40473] := 16#8770;
   // GBK_TO_UNICODE[40474] := 16#F2F2;
   // GBK_TO_UNICODE[40475] := 16#874C;
   // GBK_TO_UNICODE[40476] := 16#F2F3;
   // GBK_TO_UNICODE[40477] := 16#876E;
   // GBK_TO_UNICODE[40478] := 16#F2F4;
   // GBK_TO_UNICODE[40479] := 16#878B;
   // GBK_TO_UNICODE[40480] := 16#F2F5;
   // GBK_TO_UNICODE[40481] := 16#8753;
   // GBK_TO_UNICODE[40482] := 16#F2F6;
   // GBK_TO_UNICODE[40483] := 16#8763;
   // GBK_TO_UNICODE[40484] := 16#F2F7;
   // GBK_TO_UNICODE[40485] := 16#877C;
   // GBK_TO_UNICODE[40486] := 16#F2F8;
   // GBK_TO_UNICODE[40487] := 16#8764;
   // GBK_TO_UNICODE[40488] := 16#F2F9;
   // GBK_TO_UNICODE[40489] := 16#8759;
   // GBK_TO_UNICODE[40490] := 16#F2FA;
   // GBK_TO_UNICODE[40491] := 16#8765;
   // GBK_TO_UNICODE[40492] := 16#F2FB;
   // GBK_TO_UNICODE[40493] := 16#8793;
   // GBK_TO_UNICODE[40494] := 16#F2FC;
   // GBK_TO_UNICODE[40495] := 16#87AF;
   // GBK_TO_UNICODE[40496] := 16#F2FD;
   // GBK_TO_UNICODE[40497] := 16#87A8;
   // GBK_TO_UNICODE[40498] := 16#F2FE;
   // GBK_TO_UNICODE[40499] := 16#87D2;
   // GBK_TO_UNICODE[40500] := 16#F340;
   // GBK_TO_UNICODE[40501] := 16#9A5A;
   // GBK_TO_UNICODE[40502] := 16#F341;
   // GBK_TO_UNICODE[40503] := 16#9A5B;
   // GBK_TO_UNICODE[40504] := 16#F342;
   // GBK_TO_UNICODE[40505] := 16#9A5C;
   // GBK_TO_UNICODE[40506] := 16#F343;
   // GBK_TO_UNICODE[40507] := 16#9A5D;
   // GBK_TO_UNICODE[40508] := 16#F344;
   // GBK_TO_UNICODE[40509] := 16#9A5E;
   // GBK_TO_UNICODE[40510] := 16#F345;
   // GBK_TO_UNICODE[40511] := 16#9A5F;
   // GBK_TO_UNICODE[40512] := 16#F346;
   // GBK_TO_UNICODE[40513] := 16#9A60;
   // GBK_TO_UNICODE[40514] := 16#F347;
   // GBK_TO_UNICODE[40515] := 16#9A61;
   // GBK_TO_UNICODE[40516] := 16#F348;
   // GBK_TO_UNICODE[40517] := 16#9A62;
   // GBK_TO_UNICODE[40518] := 16#F349;
   // GBK_TO_UNICODE[40519] := 16#9A63;
   // GBK_TO_UNICODE[40520] := 16#F34A;
   // GBK_TO_UNICODE[40521] := 16#9A64;
   // GBK_TO_UNICODE[40522] := 16#F34B;
   // GBK_TO_UNICODE[40523] := 16#9A65;
   // GBK_TO_UNICODE[40524] := 16#F34C;
   // GBK_TO_UNICODE[40525] := 16#9A66;
   // GBK_TO_UNICODE[40526] := 16#F34D;
   // GBK_TO_UNICODE[40527] := 16#9A67;
   // GBK_TO_UNICODE[40528] := 16#F34E;
   // GBK_TO_UNICODE[40529] := 16#9A68;
   // GBK_TO_UNICODE[40530] := 16#F34F;
   // GBK_TO_UNICODE[40531] := 16#9A69;
   // GBK_TO_UNICODE[40532] := 16#F350;
   // GBK_TO_UNICODE[40533] := 16#9A6A;
   // GBK_TO_UNICODE[40534] := 16#F351;
   // GBK_TO_UNICODE[40535] := 16#9A6B;
   // GBK_TO_UNICODE[40536] := 16#F352;
   // GBK_TO_UNICODE[40537] := 16#9A72;
   // GBK_TO_UNICODE[40538] := 16#F353;
   // GBK_TO_UNICODE[40539] := 16#9A83;
   // GBK_TO_UNICODE[40540] := 16#F354;
   // GBK_TO_UNICODE[40541] := 16#9A89;
   // GBK_TO_UNICODE[40542] := 16#F355;
   // GBK_TO_UNICODE[40543] := 16#9A8D;
   // GBK_TO_UNICODE[40544] := 16#F356;
   // GBK_TO_UNICODE[40545] := 16#9A8E;
   // GBK_TO_UNICODE[40546] := 16#F357;
   // GBK_TO_UNICODE[40547] := 16#9A94;
   // GBK_TO_UNICODE[40548] := 16#F358;
   // GBK_TO_UNICODE[40549] := 16#9A95;
   // GBK_TO_UNICODE[40550] := 16#F359;
   // GBK_TO_UNICODE[40551] := 16#9A99;
   // GBK_TO_UNICODE[40552] := 16#F35A;
   // GBK_TO_UNICODE[40553] := 16#9AA6;
   // GBK_TO_UNICODE[40554] := 16#F35B;
   // GBK_TO_UNICODE[40555] := 16#9AA9;
   // GBK_TO_UNICODE[40556] := 16#F35C;
   // GBK_TO_UNICODE[40557] := 16#9AAA;
   // GBK_TO_UNICODE[40558] := 16#F35D;
   // GBK_TO_UNICODE[40559] := 16#9AAB;
   // GBK_TO_UNICODE[40560] := 16#F35E;
   // GBK_TO_UNICODE[40561] := 16#9AAC;
   // GBK_TO_UNICODE[40562] := 16#F35F;
   // GBK_TO_UNICODE[40563] := 16#9AAD;
   // GBK_TO_UNICODE[40564] := 16#F360;
   // GBK_TO_UNICODE[40565] := 16#9AAE;
   // GBK_TO_UNICODE[40566] := 16#F361;
   // GBK_TO_UNICODE[40567] := 16#9AAF;
   // GBK_TO_UNICODE[40568] := 16#F362;
   // GBK_TO_UNICODE[40569] := 16#9AB2;
   // GBK_TO_UNICODE[40570] := 16#F363;
   // GBK_TO_UNICODE[40571] := 16#9AB3;
   // GBK_TO_UNICODE[40572] := 16#F364;
   // GBK_TO_UNICODE[40573] := 16#9AB4;
   // GBK_TO_UNICODE[40574] := 16#F365;
   // GBK_TO_UNICODE[40575] := 16#9AB5;
   // GBK_TO_UNICODE[40576] := 16#F366;
   // GBK_TO_UNICODE[40577] := 16#9AB9;
   // GBK_TO_UNICODE[40578] := 16#F367;
   // GBK_TO_UNICODE[40579] := 16#9ABB;
   // GBK_TO_UNICODE[40580] := 16#F368;
   // GBK_TO_UNICODE[40581] := 16#9ABD;
   // GBK_TO_UNICODE[40582] := 16#F369;
   // GBK_TO_UNICODE[40583] := 16#9ABE;
   // GBK_TO_UNICODE[40584] := 16#F36A;
   // GBK_TO_UNICODE[40585] := 16#9ABF;
   // GBK_TO_UNICODE[40586] := 16#F36B;
   // GBK_TO_UNICODE[40587] := 16#9AC3;
   // GBK_TO_UNICODE[40588] := 16#F36C;
   // GBK_TO_UNICODE[40589] := 16#9AC4;
   // GBK_TO_UNICODE[40590] := 16#F36D;
   // GBK_TO_UNICODE[40591] := 16#9AC6;
   // GBK_TO_UNICODE[40592] := 16#F36E;
   // GBK_TO_UNICODE[40593] := 16#9AC7;
   // GBK_TO_UNICODE[40594] := 16#F36F;
   // GBK_TO_UNICODE[40595] := 16#9AC8;
   // GBK_TO_UNICODE[40596] := 16#F370;
   // GBK_TO_UNICODE[40597] := 16#9AC9;
   // GBK_TO_UNICODE[40598] := 16#F371;
   // GBK_TO_UNICODE[40599] := 16#9ACA;
   // GBK_TO_UNICODE[40600] := 16#F372;
   // GBK_TO_UNICODE[40601] := 16#9ACD;
   // GBK_TO_UNICODE[40602] := 16#F373;
   // GBK_TO_UNICODE[40603] := 16#9ACE;
   // GBK_TO_UNICODE[40604] := 16#F374;
   // GBK_TO_UNICODE[40605] := 16#9ACF;
   // GBK_TO_UNICODE[40606] := 16#F375;
   // GBK_TO_UNICODE[40607] := 16#9AD0;
   // GBK_TO_UNICODE[40608] := 16#F376;
   // GBK_TO_UNICODE[40609] := 16#9AD2;
   // GBK_TO_UNICODE[40610] := 16#F377;
   // GBK_TO_UNICODE[40611] := 16#9AD4;
   // GBK_TO_UNICODE[40612] := 16#F378;
   // GBK_TO_UNICODE[40613] := 16#9AD5;
   // GBK_TO_UNICODE[40614] := 16#F379;
   // GBK_TO_UNICODE[40615] := 16#9AD6;
   // GBK_TO_UNICODE[40616] := 16#F37A;
   // GBK_TO_UNICODE[40617] := 16#9AD7;
   // GBK_TO_UNICODE[40618] := 16#F37B;
   // GBK_TO_UNICODE[40619] := 16#9AD9;
   // GBK_TO_UNICODE[40620] := 16#F37C;
   // GBK_TO_UNICODE[40621] := 16#9ADA;
   // GBK_TO_UNICODE[40622] := 16#F37D;
   // GBK_TO_UNICODE[40623] := 16#9ADB;
   // GBK_TO_UNICODE[40624] := 16#F37E;
   // GBK_TO_UNICODE[40625] := 16#9ADC;
   // GBK_TO_UNICODE[40626] := 16#F380;
   // GBK_TO_UNICODE[40627] := 16#9ADD;
   // GBK_TO_UNICODE[40628] := 16#F381;
   // GBK_TO_UNICODE[40629] := 16#9ADE;
   // GBK_TO_UNICODE[40630] := 16#F382;
   // GBK_TO_UNICODE[40631] := 16#9AE0;
   // GBK_TO_UNICODE[40632] := 16#F383;
   // GBK_TO_UNICODE[40633] := 16#9AE2;
   // GBK_TO_UNICODE[40634] := 16#F384;
   // GBK_TO_UNICODE[40635] := 16#9AE3;
   // GBK_TO_UNICODE[40636] := 16#F385;
   // GBK_TO_UNICODE[40637] := 16#9AE4;
   // GBK_TO_UNICODE[40638] := 16#F386;
   // GBK_TO_UNICODE[40639] := 16#9AE5;
   // GBK_TO_UNICODE[40640] := 16#F387;
   // GBK_TO_UNICODE[40641] := 16#9AE7;
   // GBK_TO_UNICODE[40642] := 16#F388;
   // GBK_TO_UNICODE[40643] := 16#9AE8;
   // GBK_TO_UNICODE[40644] := 16#F389;
   // GBK_TO_UNICODE[40645] := 16#9AE9;
   // GBK_TO_UNICODE[40646] := 16#F38A;
   // GBK_TO_UNICODE[40647] := 16#9AEA;
   // GBK_TO_UNICODE[40648] := 16#F38B;
   // GBK_TO_UNICODE[40649] := 16#9AEC;
   // GBK_TO_UNICODE[40650] := 16#F38C;
   // GBK_TO_UNICODE[40651] := 16#9AEE;
   // GBK_TO_UNICODE[40652] := 16#F38D;
   // GBK_TO_UNICODE[40653] := 16#9AF0;
   // GBK_TO_UNICODE[40654] := 16#F38E;
   // GBK_TO_UNICODE[40655] := 16#9AF1;
   // GBK_TO_UNICODE[40656] := 16#F38F;
   // GBK_TO_UNICODE[40657] := 16#9AF2;
   // GBK_TO_UNICODE[40658] := 16#F390;
   // GBK_TO_UNICODE[40659] := 16#9AF3;
   // GBK_TO_UNICODE[40660] := 16#F391;
   // GBK_TO_UNICODE[40661] := 16#9AF4;
   // GBK_TO_UNICODE[40662] := 16#F392;
   // GBK_TO_UNICODE[40663] := 16#9AF5;
   // GBK_TO_UNICODE[40664] := 16#F393;
   // GBK_TO_UNICODE[40665] := 16#9AF6;
   // GBK_TO_UNICODE[40666] := 16#F394;
   // GBK_TO_UNICODE[40667] := 16#9AF7;
   // GBK_TO_UNICODE[40668] := 16#F395;
   // GBK_TO_UNICODE[40669] := 16#9AF8;
   // GBK_TO_UNICODE[40670] := 16#F396;
   // GBK_TO_UNICODE[40671] := 16#9AFA;
   // GBK_TO_UNICODE[40672] := 16#F397;
   // GBK_TO_UNICODE[40673] := 16#9AFC;
   // GBK_TO_UNICODE[40674] := 16#F398;
   // GBK_TO_UNICODE[40675] := 16#9AFD;
   // GBK_TO_UNICODE[40676] := 16#F399;
   // GBK_TO_UNICODE[40677] := 16#9AFE;
   // GBK_TO_UNICODE[40678] := 16#F39A;
   // GBK_TO_UNICODE[40679] := 16#9AFF;
   // GBK_TO_UNICODE[40680] := 16#F39B;
   // GBK_TO_UNICODE[40681] := 16#9B00;
   // GBK_TO_UNICODE[40682] := 16#F39C;
   // GBK_TO_UNICODE[40683] := 16#9B01;
   // GBK_TO_UNICODE[40684] := 16#F39D;
   // GBK_TO_UNICODE[40685] := 16#9B02;
   // GBK_TO_UNICODE[40686] := 16#F39E;
   // GBK_TO_UNICODE[40687] := 16#9B04;
   // GBK_TO_UNICODE[40688] := 16#F39F;
   // GBK_TO_UNICODE[40689] := 16#9B05;
   // GBK_TO_UNICODE[40690] := 16#F3A0;
   // GBK_TO_UNICODE[40691] := 16#9B06;
   // GBK_TO_UNICODE[40692] := 16#F3A1;
   // GBK_TO_UNICODE[40693] := 16#87C6;
   // GBK_TO_UNICODE[40694] := 16#F3A2;
   // GBK_TO_UNICODE[40695] := 16#8788;
   // GBK_TO_UNICODE[40696] := 16#F3A3;
   // GBK_TO_UNICODE[40697] := 16#8785;
   // GBK_TO_UNICODE[40698] := 16#F3A4;
   // GBK_TO_UNICODE[40699] := 16#87AD;
   // GBK_TO_UNICODE[40700] := 16#F3A5;
   // GBK_TO_UNICODE[40701] := 16#8797;
   // GBK_TO_UNICODE[40702] := 16#F3A6;
   // GBK_TO_UNICODE[40703] := 16#8783;
   // GBK_TO_UNICODE[40704] := 16#F3A7;
   // GBK_TO_UNICODE[40705] := 16#87AB;
   // GBK_TO_UNICODE[40706] := 16#F3A8;
   // GBK_TO_UNICODE[40707] := 16#87E5;
   // GBK_TO_UNICODE[40708] := 16#F3A9;
   // GBK_TO_UNICODE[40709] := 16#87AC;
   // GBK_TO_UNICODE[40710] := 16#F3AA;
   // GBK_TO_UNICODE[40711] := 16#87B5;
   // GBK_TO_UNICODE[40712] := 16#F3AB;
   // GBK_TO_UNICODE[40713] := 16#87B3;
   // GBK_TO_UNICODE[40714] := 16#F3AC;
   // GBK_TO_UNICODE[40715] := 16#87CB;
   // GBK_TO_UNICODE[40716] := 16#F3AD;
   // GBK_TO_UNICODE[40717] := 16#87D3;
   // GBK_TO_UNICODE[40718] := 16#F3AE;
   // GBK_TO_UNICODE[40719] := 16#87BD;
   // GBK_TO_UNICODE[40720] := 16#F3AF;
   // GBK_TO_UNICODE[40721] := 16#87D1;
   // GBK_TO_UNICODE[40722] := 16#F3B0;
   // GBK_TO_UNICODE[40723] := 16#87C0;
   // GBK_TO_UNICODE[40724] := 16#F3B1;
   // GBK_TO_UNICODE[40725] := 16#87CA;
   // GBK_TO_UNICODE[40726] := 16#F3B2;
   // GBK_TO_UNICODE[40727] := 16#87DB;
   // GBK_TO_UNICODE[40728] := 16#F3B3;
   // GBK_TO_UNICODE[40729] := 16#87EA;
   // GBK_TO_UNICODE[40730] := 16#F3B4;
   // GBK_TO_UNICODE[40731] := 16#87E0;
   // GBK_TO_UNICODE[40732] := 16#F3B5;
   // GBK_TO_UNICODE[40733] := 16#87EE;
   // GBK_TO_UNICODE[40734] := 16#F3B6;
   // GBK_TO_UNICODE[40735] := 16#8816;
   // GBK_TO_UNICODE[40736] := 16#F3B7;
   // GBK_TO_UNICODE[40737] := 16#8813;
   // GBK_TO_UNICODE[40738] := 16#F3B8;
   // GBK_TO_UNICODE[40739] := 16#87FE;
   // GBK_TO_UNICODE[40740] := 16#F3B9;
   // GBK_TO_UNICODE[40741] := 16#880A;
   // GBK_TO_UNICODE[40742] := 16#F3BA;
   // GBK_TO_UNICODE[40743] := 16#881B;
   // GBK_TO_UNICODE[40744] := 16#F3BB;
   // GBK_TO_UNICODE[40745] := 16#8821;
   // GBK_TO_UNICODE[40746] := 16#F3BC;
   // GBK_TO_UNICODE[40747] := 16#8839;
   // GBK_TO_UNICODE[40748] := 16#F3BD;
   // GBK_TO_UNICODE[40749] := 16#883C;
   // GBK_TO_UNICODE[40750] := 16#F3BE;
   // GBK_TO_UNICODE[40751] := 16#7F36;
   // GBK_TO_UNICODE[40752] := 16#F3BF;
   // GBK_TO_UNICODE[40753] := 16#7F42;
   // GBK_TO_UNICODE[40754] := 16#F3C0;
   // GBK_TO_UNICODE[40755] := 16#7F44;
   // GBK_TO_UNICODE[40756] := 16#F3C1;
   // GBK_TO_UNICODE[40757] := 16#7F45;
   // GBK_TO_UNICODE[40758] := 16#F3C2;
   // GBK_TO_UNICODE[40759] := 16#8210;
   // GBK_TO_UNICODE[40760] := 16#F3C3;
   // GBK_TO_UNICODE[40761] := 16#7AFA;
   // GBK_TO_UNICODE[40762] := 16#F3C4;
   // GBK_TO_UNICODE[40763] := 16#7AFD;
   // GBK_TO_UNICODE[40764] := 16#F3C5;
   // GBK_TO_UNICODE[40765] := 16#7B08;
   // GBK_TO_UNICODE[40766] := 16#F3C6;
   // GBK_TO_UNICODE[40767] := 16#7B03;
   // GBK_TO_UNICODE[40768] := 16#F3C7;
   // GBK_TO_UNICODE[40769] := 16#7B04;
   // GBK_TO_UNICODE[40770] := 16#F3C8;
   // GBK_TO_UNICODE[40771] := 16#7B15;
   // GBK_TO_UNICODE[40772] := 16#F3C9;
   // GBK_TO_UNICODE[40773] := 16#7B0A;
   // GBK_TO_UNICODE[40774] := 16#F3CA;
   // GBK_TO_UNICODE[40775] := 16#7B2B;
   // GBK_TO_UNICODE[40776] := 16#F3CB;
   // GBK_TO_UNICODE[40777] := 16#7B0F;
   // GBK_TO_UNICODE[40778] := 16#F3CC;
   // GBK_TO_UNICODE[40779] := 16#7B47;
   // GBK_TO_UNICODE[40780] := 16#F3CD;
   // GBK_TO_UNICODE[40781] := 16#7B38;
   // GBK_TO_UNICODE[40782] := 16#F3CE;
   // GBK_TO_UNICODE[40783] := 16#7B2A;
   // GBK_TO_UNICODE[40784] := 16#F3CF;
   // GBK_TO_UNICODE[40785] := 16#7B19;
   // GBK_TO_UNICODE[40786] := 16#F3D0;
   // GBK_TO_UNICODE[40787] := 16#7B2E;
   // GBK_TO_UNICODE[40788] := 16#F3D1;
   // GBK_TO_UNICODE[40789] := 16#7B31;
   // GBK_TO_UNICODE[40790] := 16#F3D2;
   // GBK_TO_UNICODE[40791] := 16#7B20;
   // GBK_TO_UNICODE[40792] := 16#F3D3;
   // GBK_TO_UNICODE[40793] := 16#7B25;
   // GBK_TO_UNICODE[40794] := 16#F3D4;
   // GBK_TO_UNICODE[40795] := 16#7B24;
   // GBK_TO_UNICODE[40796] := 16#F3D5;
   // GBK_TO_UNICODE[40797] := 16#7B33;
   // GBK_TO_UNICODE[40798] := 16#F3D6;
   // GBK_TO_UNICODE[40799] := 16#7B3E;
   // GBK_TO_UNICODE[40800] := 16#F3D7;
   // GBK_TO_UNICODE[40801] := 16#7B1E;
   // GBK_TO_UNICODE[40802] := 16#F3D8;
   // GBK_TO_UNICODE[40803] := 16#7B58;
   // GBK_TO_UNICODE[40804] := 16#F3D9;
   // GBK_TO_UNICODE[40805] := 16#7B5A;
   // GBK_TO_UNICODE[40806] := 16#F3DA;
   // GBK_TO_UNICODE[40807] := 16#7B45;
   // GBK_TO_UNICODE[40808] := 16#F3DB;
   // GBK_TO_UNICODE[40809] := 16#7B75;
   // GBK_TO_UNICODE[40810] := 16#F3DC;
   // GBK_TO_UNICODE[40811] := 16#7B4C;
   // GBK_TO_UNICODE[40812] := 16#F3DD;
   // GBK_TO_UNICODE[40813] := 16#7B5D;
   // GBK_TO_UNICODE[40814] := 16#F3DE;
   // GBK_TO_UNICODE[40815] := 16#7B60;
   // GBK_TO_UNICODE[40816] := 16#F3DF;
   // GBK_TO_UNICODE[40817] := 16#7B6E;
   // GBK_TO_UNICODE[40818] := 16#F3E0;
   // GBK_TO_UNICODE[40819] := 16#7B7B;
   // GBK_TO_UNICODE[40820] := 16#F3E1;
   // GBK_TO_UNICODE[40821] := 16#7B62;
   // GBK_TO_UNICODE[40822] := 16#F3E2;
   // GBK_TO_UNICODE[40823] := 16#7B72;
   // GBK_TO_UNICODE[40824] := 16#F3E3;
   // GBK_TO_UNICODE[40825] := 16#7B71;
   // GBK_TO_UNICODE[40826] := 16#F3E4;
   // GBK_TO_UNICODE[40827] := 16#7B90;
   // GBK_TO_UNICODE[40828] := 16#F3E5;
   // GBK_TO_UNICODE[40829] := 16#7BA6;
   // GBK_TO_UNICODE[40830] := 16#F3E6;
   // GBK_TO_UNICODE[40831] := 16#7BA7;
   // GBK_TO_UNICODE[40832] := 16#F3E7;
   // GBK_TO_UNICODE[40833] := 16#7BB8;
   // GBK_TO_UNICODE[40834] := 16#F3E8;
   // GBK_TO_UNICODE[40835] := 16#7BAC;
   // GBK_TO_UNICODE[40836] := 16#F3E9;
   // GBK_TO_UNICODE[40837] := 16#7B9D;
   // GBK_TO_UNICODE[40838] := 16#F3EA;
   // GBK_TO_UNICODE[40839] := 16#7BA8;
   // GBK_TO_UNICODE[40840] := 16#F3EB;
   // GBK_TO_UNICODE[40841] := 16#7B85;
   // GBK_TO_UNICODE[40842] := 16#F3EC;
   // GBK_TO_UNICODE[40843] := 16#7BAA;
   // GBK_TO_UNICODE[40844] := 16#F3ED;
   // GBK_TO_UNICODE[40845] := 16#7B9C;
   // GBK_TO_UNICODE[40846] := 16#F3EE;
   // GBK_TO_UNICODE[40847] := 16#7BA2;
   // GBK_TO_UNICODE[40848] := 16#F3EF;
   // GBK_TO_UNICODE[40849] := 16#7BAB;
   // GBK_TO_UNICODE[40850] := 16#F3F0;
   // GBK_TO_UNICODE[40851] := 16#7BB4;
   // GBK_TO_UNICODE[40852] := 16#F3F1;
   // GBK_TO_UNICODE[40853] := 16#7BD1;
   // GBK_TO_UNICODE[40854] := 16#F3F2;
   // GBK_TO_UNICODE[40855] := 16#7BC1;
   // GBK_TO_UNICODE[40856] := 16#F3F3;
   // GBK_TO_UNICODE[40857] := 16#7BCC;
   // GBK_TO_UNICODE[40858] := 16#F3F4;
   // GBK_TO_UNICODE[40859] := 16#7BDD;
   // GBK_TO_UNICODE[40860] := 16#F3F5;
   // GBK_TO_UNICODE[40861] := 16#7BDA;
   // GBK_TO_UNICODE[40862] := 16#F3F6;
   // GBK_TO_UNICODE[40863] := 16#7BE5;
   // GBK_TO_UNICODE[40864] := 16#F3F7;
   // GBK_TO_UNICODE[40865] := 16#7BE6;
   // GBK_TO_UNICODE[40866] := 16#F3F8;
   // GBK_TO_UNICODE[40867] := 16#7BEA;
   // GBK_TO_UNICODE[40868] := 16#F3F9;
   // GBK_TO_UNICODE[40869] := 16#7C0C;
   // GBK_TO_UNICODE[40870] := 16#F3FA;
   // GBK_TO_UNICODE[40871] := 16#7BFE;
   // GBK_TO_UNICODE[40872] := 16#F3FB;
   // GBK_TO_UNICODE[40873] := 16#7BFC;
   // GBK_TO_UNICODE[40874] := 16#F3FC;
   // GBK_TO_UNICODE[40875] := 16#7C0F;
   // GBK_TO_UNICODE[40876] := 16#F3FD;
   // GBK_TO_UNICODE[40877] := 16#7C16;
   // GBK_TO_UNICODE[40878] := 16#F3FE;
   // GBK_TO_UNICODE[40879] := 16#7C0B;
   // GBK_TO_UNICODE[40880] := 16#F440;
   // GBK_TO_UNICODE[40881] := 16#9B07;
   // GBK_TO_UNICODE[40882] := 16#F441;
   // GBK_TO_UNICODE[40883] := 16#9B09;
   // GBK_TO_UNICODE[40884] := 16#F442;
   // GBK_TO_UNICODE[40885] := 16#9B0A;
   // GBK_TO_UNICODE[40886] := 16#F443;
   // GBK_TO_UNICODE[40887] := 16#9B0B;
   // GBK_TO_UNICODE[40888] := 16#F444;
   // GBK_TO_UNICODE[40889] := 16#9B0C;
   // GBK_TO_UNICODE[40890] := 16#F445;
   // GBK_TO_UNICODE[40891] := 16#9B0D;
   // GBK_TO_UNICODE[40892] := 16#F446;
   // GBK_TO_UNICODE[40893] := 16#9B0E;
   // GBK_TO_UNICODE[40894] := 16#F447;
   // GBK_TO_UNICODE[40895] := 16#9B10;
   // GBK_TO_UNICODE[40896] := 16#F448;
   // GBK_TO_UNICODE[40897] := 16#9B11;
   // GBK_TO_UNICODE[40898] := 16#F449;
   // GBK_TO_UNICODE[40899] := 16#9B12;
   // GBK_TO_UNICODE[40900] := 16#F44A;
   // GBK_TO_UNICODE[40901] := 16#9B14;
   // GBK_TO_UNICODE[40902] := 16#F44B;
   // GBK_TO_UNICODE[40903] := 16#9B15;
   // GBK_TO_UNICODE[40904] := 16#F44C;
   // GBK_TO_UNICODE[40905] := 16#9B16;
   // GBK_TO_UNICODE[40906] := 16#F44D;
   // GBK_TO_UNICODE[40907] := 16#9B17;
   // GBK_TO_UNICODE[40908] := 16#F44E;
   // GBK_TO_UNICODE[40909] := 16#9B18;
   // GBK_TO_UNICODE[40910] := 16#F44F;
   // GBK_TO_UNICODE[40911] := 16#9B19;
   // GBK_TO_UNICODE[40912] := 16#F450;
   // GBK_TO_UNICODE[40913] := 16#9B1A;
   // GBK_TO_UNICODE[40914] := 16#F451;
   // GBK_TO_UNICODE[40915] := 16#9B1B;
   // GBK_TO_UNICODE[40916] := 16#F452;
   // GBK_TO_UNICODE[40917] := 16#9B1C;
   // GBK_TO_UNICODE[40918] := 16#F453;
   // GBK_TO_UNICODE[40919] := 16#9B1D;
   // GBK_TO_UNICODE[40920] := 16#F454;
   // GBK_TO_UNICODE[40921] := 16#9B1E;
   // GBK_TO_UNICODE[40922] := 16#F455;
   // GBK_TO_UNICODE[40923] := 16#9B20;
   // GBK_TO_UNICODE[40924] := 16#F456;
   // GBK_TO_UNICODE[40925] := 16#9B21;
   // GBK_TO_UNICODE[40926] := 16#F457;
   // GBK_TO_UNICODE[40927] := 16#9B22;
   // GBK_TO_UNICODE[40928] := 16#F458;
   // GBK_TO_UNICODE[40929] := 16#9B24;
   // GBK_TO_UNICODE[40930] := 16#F459;
   // GBK_TO_UNICODE[40931] := 16#9B25;
   // GBK_TO_UNICODE[40932] := 16#F45A;
   // GBK_TO_UNICODE[40933] := 16#9B26;
   // GBK_TO_UNICODE[40934] := 16#F45B;
   // GBK_TO_UNICODE[40935] := 16#9B27;
   // GBK_TO_UNICODE[40936] := 16#F45C;
   // GBK_TO_UNICODE[40937] := 16#9B28;
   // GBK_TO_UNICODE[40938] := 16#F45D;
   // GBK_TO_UNICODE[40939] := 16#9B29;
   // GBK_TO_UNICODE[40940] := 16#F45E;
   // GBK_TO_UNICODE[40941] := 16#9B2A;
   // GBK_TO_UNICODE[40942] := 16#F45F;
   // GBK_TO_UNICODE[40943] := 16#9B2B;
   // GBK_TO_UNICODE[40944] := 16#F460;
   // GBK_TO_UNICODE[40945] := 16#9B2C;
   // GBK_TO_UNICODE[40946] := 16#F461;
   // GBK_TO_UNICODE[40947] := 16#9B2D;
   // GBK_TO_UNICODE[40948] := 16#F462;
   // GBK_TO_UNICODE[40949] := 16#9B2E;
   // GBK_TO_UNICODE[40950] := 16#F463;
   // GBK_TO_UNICODE[40951] := 16#9B30;
   // GBK_TO_UNICODE[40952] := 16#F464;
   // GBK_TO_UNICODE[40953] := 16#9B31;
   // GBK_TO_UNICODE[40954] := 16#F465;
   // GBK_TO_UNICODE[40955] := 16#9B33;
   // GBK_TO_UNICODE[40956] := 16#F466;
   // GBK_TO_UNICODE[40957] := 16#9B34;
   // GBK_TO_UNICODE[40958] := 16#F467;
   // GBK_TO_UNICODE[40959] := 16#9B35;
   // GBK_TO_UNICODE[40960] := 16#F468;
   // GBK_TO_UNICODE[40961] := 16#9B36;
   // GBK_TO_UNICODE[40962] := 16#F469;
   // GBK_TO_UNICODE[40963] := 16#9B37;
   // GBK_TO_UNICODE[40964] := 16#F46A;
   // GBK_TO_UNICODE[40965] := 16#9B38;
   // GBK_TO_UNICODE[40966] := 16#F46B;
   // GBK_TO_UNICODE[40967] := 16#9B39;
   // GBK_TO_UNICODE[40968] := 16#F46C;
   // GBK_TO_UNICODE[40969] := 16#9B3A;
   // GBK_TO_UNICODE[40970] := 16#F46D;
   // GBK_TO_UNICODE[40971] := 16#9B3D;
   // GBK_TO_UNICODE[40972] := 16#F46E;
   // GBK_TO_UNICODE[40973] := 16#9B3E;
   // GBK_TO_UNICODE[40974] := 16#F46F;
   // GBK_TO_UNICODE[40975] := 16#9B3F;
   // GBK_TO_UNICODE[40976] := 16#F470;
   // GBK_TO_UNICODE[40977] := 16#9B40;
   // GBK_TO_UNICODE[40978] := 16#F471;
   // GBK_TO_UNICODE[40979] := 16#9B46;
   // GBK_TO_UNICODE[40980] := 16#F472;
   // GBK_TO_UNICODE[40981] := 16#9B4A;
   // GBK_TO_UNICODE[40982] := 16#F473;
   // GBK_TO_UNICODE[40983] := 16#9B4B;
   // GBK_TO_UNICODE[40984] := 16#F474;
   // GBK_TO_UNICODE[40985] := 16#9B4C;
   // GBK_TO_UNICODE[40986] := 16#F475;
   // GBK_TO_UNICODE[40987] := 16#9B4E;
   // GBK_TO_UNICODE[40988] := 16#F476;
   // GBK_TO_UNICODE[40989] := 16#9B50;
   // GBK_TO_UNICODE[40990] := 16#F477;
   // GBK_TO_UNICODE[40991] := 16#9B52;
   // GBK_TO_UNICODE[40992] := 16#F478;
   // GBK_TO_UNICODE[40993] := 16#9B53;
   // GBK_TO_UNICODE[40994] := 16#F479;
   // GBK_TO_UNICODE[40995] := 16#9B55;
   // GBK_TO_UNICODE[40996] := 16#F47A;
   // GBK_TO_UNICODE[40997] := 16#9B56;
   // GBK_TO_UNICODE[40998] := 16#F47B;
   // GBK_TO_UNICODE[40999] := 16#9B57;
   // GBK_TO_UNICODE[41000] := 16#F47C;
   // GBK_TO_UNICODE[41001] := 16#9B58;
   // GBK_TO_UNICODE[41002] := 16#F47D;
   // GBK_TO_UNICODE[41003] := 16#9B59;
   // GBK_TO_UNICODE[41004] := 16#F47E;
   // GBK_TO_UNICODE[41005] := 16#9B5A;
   // GBK_TO_UNICODE[41006] := 16#F480;
   // GBK_TO_UNICODE[41007] := 16#9B5B;
   // GBK_TO_UNICODE[41008] := 16#F481;
   // GBK_TO_UNICODE[41009] := 16#9B5C;
   // GBK_TO_UNICODE[41010] := 16#F482;
   // GBK_TO_UNICODE[41011] := 16#9B5D;
   // GBK_TO_UNICODE[41012] := 16#F483;
   // GBK_TO_UNICODE[41013] := 16#9B5E;
   // GBK_TO_UNICODE[41014] := 16#F484;
   // GBK_TO_UNICODE[41015] := 16#9B5F;
   // GBK_TO_UNICODE[41016] := 16#F485;
   // GBK_TO_UNICODE[41017] := 16#9B60;
   // GBK_TO_UNICODE[41018] := 16#F486;
   // GBK_TO_UNICODE[41019] := 16#9B61;
   // GBK_TO_UNICODE[41020] := 16#F487;
   // GBK_TO_UNICODE[41021] := 16#9B62;
   // GBK_TO_UNICODE[41022] := 16#F488;
   // GBK_TO_UNICODE[41023] := 16#9B63;
   // GBK_TO_UNICODE[41024] := 16#F489;
   // GBK_TO_UNICODE[41025] := 16#9B64;
   // GBK_TO_UNICODE[41026] := 16#F48A;
   // GBK_TO_UNICODE[41027] := 16#9B65;
   // GBK_TO_UNICODE[41028] := 16#F48B;
   // GBK_TO_UNICODE[41029] := 16#9B66;
   // GBK_TO_UNICODE[41030] := 16#F48C;
   // GBK_TO_UNICODE[41031] := 16#9B67;
   // GBK_TO_UNICODE[41032] := 16#F48D;
   // GBK_TO_UNICODE[41033] := 16#9B68;
   // GBK_TO_UNICODE[41034] := 16#F48E;
   // GBK_TO_UNICODE[41035] := 16#9B69;
   // GBK_TO_UNICODE[41036] := 16#F48F;
   // GBK_TO_UNICODE[41037] := 16#9B6A;
   // GBK_TO_UNICODE[41038] := 16#F490;
   // GBK_TO_UNICODE[41039] := 16#9B6B;
   // GBK_TO_UNICODE[41040] := 16#F491;
   // GBK_TO_UNICODE[41041] := 16#9B6C;
   // GBK_TO_UNICODE[41042] := 16#F492;
   // GBK_TO_UNICODE[41043] := 16#9B6D;
   // GBK_TO_UNICODE[41044] := 16#F493;
   // GBK_TO_UNICODE[41045] := 16#9B6E;
   // GBK_TO_UNICODE[41046] := 16#F494;
   // GBK_TO_UNICODE[41047] := 16#9B6F;
   // GBK_TO_UNICODE[41048] := 16#F495;
   // GBK_TO_UNICODE[41049] := 16#9B70;
   // GBK_TO_UNICODE[41050] := 16#F496;
   // GBK_TO_UNICODE[41051] := 16#9B71;
   // GBK_TO_UNICODE[41052] := 16#F497;
   // GBK_TO_UNICODE[41053] := 16#9B72;
   // GBK_TO_UNICODE[41054] := 16#F498;
   // GBK_TO_UNICODE[41055] := 16#9B73;
   // GBK_TO_UNICODE[41056] := 16#F499;
   // GBK_TO_UNICODE[41057] := 16#9B74;
   // GBK_TO_UNICODE[41058] := 16#F49A;
   // GBK_TO_UNICODE[41059] := 16#9B75;
   // GBK_TO_UNICODE[41060] := 16#F49B;
   // GBK_TO_UNICODE[41061] := 16#9B76;
   // GBK_TO_UNICODE[41062] := 16#F49C;
   // GBK_TO_UNICODE[41063] := 16#9B77;
   // GBK_TO_UNICODE[41064] := 16#F49D;
   // GBK_TO_UNICODE[41065] := 16#9B78;
   // GBK_TO_UNICODE[41066] := 16#F49E;
   // GBK_TO_UNICODE[41067] := 16#9B79;
   // GBK_TO_UNICODE[41068] := 16#F49F;
   // GBK_TO_UNICODE[41069] := 16#9B7A;
   // GBK_TO_UNICODE[41070] := 16#F4A0;
   // GBK_TO_UNICODE[41071] := 16#9B7B;
   // GBK_TO_UNICODE[41072] := 16#F4A1;
   // GBK_TO_UNICODE[41073] := 16#7C1F;
   // GBK_TO_UNICODE[41074] := 16#F4A2;
   // GBK_TO_UNICODE[41075] := 16#7C2A;
   // GBK_TO_UNICODE[41076] := 16#F4A3;
   // GBK_TO_UNICODE[41077] := 16#7C26;
   // GBK_TO_UNICODE[41078] := 16#F4A4;
   // GBK_TO_UNICODE[41079] := 16#7C38;
   // GBK_TO_UNICODE[41080] := 16#F4A5;
   // GBK_TO_UNICODE[41081] := 16#7C41;
   // GBK_TO_UNICODE[41082] := 16#F4A6;
   // GBK_TO_UNICODE[41083] := 16#7C40;
   // GBK_TO_UNICODE[41084] := 16#F4A7;
   // GBK_TO_UNICODE[41085] := 16#81FE;
   // GBK_TO_UNICODE[41086] := 16#F4A8;
   // GBK_TO_UNICODE[41087] := 16#8201;
   // GBK_TO_UNICODE[41088] := 16#F4A9;
   // GBK_TO_UNICODE[41089] := 16#8202;
   // GBK_TO_UNICODE[41090] := 16#F4AA;
   // GBK_TO_UNICODE[41091] := 16#8204;
   // GBK_TO_UNICODE[41092] := 16#F4AB;
   // GBK_TO_UNICODE[41093] := 16#81EC;
   // GBK_TO_UNICODE[41094] := 16#F4AC;
   // GBK_TO_UNICODE[41095] := 16#8844;
   // GBK_TO_UNICODE[41096] := 16#F4AD;
   // GBK_TO_UNICODE[41097] := 16#8221;
   // GBK_TO_UNICODE[41098] := 16#F4AE;
   // GBK_TO_UNICODE[41099] := 16#8222;
   // GBK_TO_UNICODE[41100] := 16#F4AF;
   // GBK_TO_UNICODE[41101] := 16#8223;
   // GBK_TO_UNICODE[41102] := 16#F4B0;
   // GBK_TO_UNICODE[41103] := 16#822D;
   // GBK_TO_UNICODE[41104] := 16#F4B1;
   // GBK_TO_UNICODE[41105] := 16#822F;
   // GBK_TO_UNICODE[41106] := 16#F4B2;
   // GBK_TO_UNICODE[41107] := 16#8228;
   // GBK_TO_UNICODE[41108] := 16#F4B3;
   // GBK_TO_UNICODE[41109] := 16#822B;
   // GBK_TO_UNICODE[41110] := 16#F4B4;
   // GBK_TO_UNICODE[41111] := 16#8238;
   // GBK_TO_UNICODE[41112] := 16#F4B5;
   // GBK_TO_UNICODE[41113] := 16#823B;
   // GBK_TO_UNICODE[41114] := 16#F4B6;
   // GBK_TO_UNICODE[41115] := 16#8233;
   // GBK_TO_UNICODE[41116] := 16#F4B7;
   // GBK_TO_UNICODE[41117] := 16#8234;
   // GBK_TO_UNICODE[41118] := 16#F4B8;
   // GBK_TO_UNICODE[41119] := 16#823E;
   // GBK_TO_UNICODE[41120] := 16#F4B9;
   // GBK_TO_UNICODE[41121] := 16#8244;
   // GBK_TO_UNICODE[41122] := 16#F4BA;
   // GBK_TO_UNICODE[41123] := 16#8249;
   // GBK_TO_UNICODE[41124] := 16#F4BB;
   // GBK_TO_UNICODE[41125] := 16#824B;
   // GBK_TO_UNICODE[41126] := 16#F4BC;
   // GBK_TO_UNICODE[41127] := 16#824F;
   // GBK_TO_UNICODE[41128] := 16#F4BD;
   // GBK_TO_UNICODE[41129] := 16#825A;
   // GBK_TO_UNICODE[41130] := 16#F4BE;
   // GBK_TO_UNICODE[41131] := 16#825F;
   // GBK_TO_UNICODE[41132] := 16#F4BF;
   // GBK_TO_UNICODE[41133] := 16#8268;
   // GBK_TO_UNICODE[41134] := 16#F4C0;
   // GBK_TO_UNICODE[41135] := 16#887E;
   // GBK_TO_UNICODE[41136] := 16#F4C1;
   // GBK_TO_UNICODE[41137] := 16#8885;
   // GBK_TO_UNICODE[41138] := 16#F4C2;
   // GBK_TO_UNICODE[41139] := 16#8888;
   // GBK_TO_UNICODE[41140] := 16#F4C3;
   // GBK_TO_UNICODE[41141] := 16#88D8;
   // GBK_TO_UNICODE[41142] := 16#F4C4;
   // GBK_TO_UNICODE[41143] := 16#88DF;
   // GBK_TO_UNICODE[41144] := 16#F4C5;
   // GBK_TO_UNICODE[41145] := 16#895E;
   // GBK_TO_UNICODE[41146] := 16#F4C6;
   // GBK_TO_UNICODE[41147] := 16#7F9D;
   // GBK_TO_UNICODE[41148] := 16#F4C7;
   // GBK_TO_UNICODE[41149] := 16#7F9F;
   // GBK_TO_UNICODE[41150] := 16#F4C8;
   // GBK_TO_UNICODE[41151] := 16#7FA7;
   // GBK_TO_UNICODE[41152] := 16#F4C9;
   // GBK_TO_UNICODE[41153] := 16#7FAF;
   // GBK_TO_UNICODE[41154] := 16#F4CA;
   // GBK_TO_UNICODE[41155] := 16#7FB0;
   // GBK_TO_UNICODE[41156] := 16#F4CB;
   // GBK_TO_UNICODE[41157] := 16#7FB2;
   // GBK_TO_UNICODE[41158] := 16#F4CC;
   // GBK_TO_UNICODE[41159] := 16#7C7C;
   // GBK_TO_UNICODE[41160] := 16#F4CD;
   // GBK_TO_UNICODE[41161] := 16#6549;
   // GBK_TO_UNICODE[41162] := 16#F4CE;
   // GBK_TO_UNICODE[41163] := 16#7C91;
   // GBK_TO_UNICODE[41164] := 16#F4CF;
   // GBK_TO_UNICODE[41165] := 16#7C9D;
   // GBK_TO_UNICODE[41166] := 16#F4D0;
   // GBK_TO_UNICODE[41167] := 16#7C9C;
   // GBK_TO_UNICODE[41168] := 16#F4D1;
   // GBK_TO_UNICODE[41169] := 16#7C9E;
   // GBK_TO_UNICODE[41170] := 16#F4D2;
   // GBK_TO_UNICODE[41171] := 16#7CA2;
   // GBK_TO_UNICODE[41172] := 16#F4D3;
   // GBK_TO_UNICODE[41173] := 16#7CB2;
   // GBK_TO_UNICODE[41174] := 16#F4D4;
   // GBK_TO_UNICODE[41175] := 16#7CBC;
   // GBK_TO_UNICODE[41176] := 16#F4D5;
   // GBK_TO_UNICODE[41177] := 16#7CBD;
   // GBK_TO_UNICODE[41178] := 16#F4D6;
   // GBK_TO_UNICODE[41179] := 16#7CC1;
   // GBK_TO_UNICODE[41180] := 16#F4D7;
   // GBK_TO_UNICODE[41181] := 16#7CC7;
   // GBK_TO_UNICODE[41182] := 16#F4D8;
   // GBK_TO_UNICODE[41183] := 16#7CCC;
   // GBK_TO_UNICODE[41184] := 16#F4D9;
   // GBK_TO_UNICODE[41185] := 16#7CCD;
   // GBK_TO_UNICODE[41186] := 16#F4DA;
   // GBK_TO_UNICODE[41187] := 16#7CC8;
   // GBK_TO_UNICODE[41188] := 16#F4DB;
   // GBK_TO_UNICODE[41189] := 16#7CC5;
   // GBK_TO_UNICODE[41190] := 16#F4DC;
   // GBK_TO_UNICODE[41191] := 16#7CD7;
   // GBK_TO_UNICODE[41192] := 16#F4DD;
   // GBK_TO_UNICODE[41193] := 16#7CE8;
   // GBK_TO_UNICODE[41194] := 16#F4DE;
   // GBK_TO_UNICODE[41195] := 16#826E;
   // GBK_TO_UNICODE[41196] := 16#F4DF;
   // GBK_TO_UNICODE[41197] := 16#66A8;
   // GBK_TO_UNICODE[41198] := 16#F4E0;
   // GBK_TO_UNICODE[41199] := 16#7FBF;
   // GBK_TO_UNICODE[41200] := 16#F4E1;
   // GBK_TO_UNICODE[41201] := 16#7FCE;
   // GBK_TO_UNICODE[41202] := 16#F4E2;
   // GBK_TO_UNICODE[41203] := 16#7FD5;
   // GBK_TO_UNICODE[41204] := 16#F4E3;
   // GBK_TO_UNICODE[41205] := 16#7FE5;
   // GBK_TO_UNICODE[41206] := 16#F4E4;
   // GBK_TO_UNICODE[41207] := 16#7FE1;
   // GBK_TO_UNICODE[41208] := 16#F4E5;
   // GBK_TO_UNICODE[41209] := 16#7FE6;
   // GBK_TO_UNICODE[41210] := 16#F4E6;
   // GBK_TO_UNICODE[41211] := 16#7FE9;
   // GBK_TO_UNICODE[41212] := 16#F4E7;
   // GBK_TO_UNICODE[41213] := 16#7FEE;
   // GBK_TO_UNICODE[41214] := 16#F4E8;
   // GBK_TO_UNICODE[41215] := 16#7FF3;
   // GBK_TO_UNICODE[41216] := 16#F4E9;
   // GBK_TO_UNICODE[41217] := 16#7CF8;
   // GBK_TO_UNICODE[41218] := 16#F4EA;
   // GBK_TO_UNICODE[41219] := 16#7D77;
   // GBK_TO_UNICODE[41220] := 16#F4EB;
   // GBK_TO_UNICODE[41221] := 16#7DA6;
   // GBK_TO_UNICODE[41222] := 16#F4EC;
   // GBK_TO_UNICODE[41223] := 16#7DAE;
   // GBK_TO_UNICODE[41224] := 16#F4ED;
   // GBK_TO_UNICODE[41225] := 16#7E47;
   // GBK_TO_UNICODE[41226] := 16#F4EE;
   // GBK_TO_UNICODE[41227] := 16#7E9B;
   // GBK_TO_UNICODE[41228] := 16#F4EF;
   // GBK_TO_UNICODE[41229] := 16#9EB8;
   // GBK_TO_UNICODE[41230] := 16#F4F0;
   // GBK_TO_UNICODE[41231] := 16#9EB4;
   // GBK_TO_UNICODE[41232] := 16#F4F1;
   // GBK_TO_UNICODE[41233] := 16#8D73;
   // GBK_TO_UNICODE[41234] := 16#F4F2;
   // GBK_TO_UNICODE[41235] := 16#8D84;
   // GBK_TO_UNICODE[41236] := 16#F4F3;
   // GBK_TO_UNICODE[41237] := 16#8D94;
   // GBK_TO_UNICODE[41238] := 16#F4F4;
   // GBK_TO_UNICODE[41239] := 16#8D91;
   // GBK_TO_UNICODE[41240] := 16#F4F5;
   // GBK_TO_UNICODE[41241] := 16#8DB1;
   // GBK_TO_UNICODE[41242] := 16#F4F6;
   // GBK_TO_UNICODE[41243] := 16#8D67;
   // GBK_TO_UNICODE[41244] := 16#F4F7;
   // GBK_TO_UNICODE[41245] := 16#8D6D;
   // GBK_TO_UNICODE[41246] := 16#F4F8;
   // GBK_TO_UNICODE[41247] := 16#8C47;
   // GBK_TO_UNICODE[41248] := 16#F4F9;
   // GBK_TO_UNICODE[41249] := 16#8C49;
   // GBK_TO_UNICODE[41250] := 16#F4FA;
   // GBK_TO_UNICODE[41251] := 16#914A;
   // GBK_TO_UNICODE[41252] := 16#F4FB;
   // GBK_TO_UNICODE[41253] := 16#9150;
   // GBK_TO_UNICODE[41254] := 16#F4FC;
   // GBK_TO_UNICODE[41255] := 16#914E;
   // GBK_TO_UNICODE[41256] := 16#F4FD;
   // GBK_TO_UNICODE[41257] := 16#914F;
   // GBK_TO_UNICODE[41258] := 16#F4FE;
   // GBK_TO_UNICODE[41259] := 16#9164;
   // GBK_TO_UNICODE[41260] := 16#F540;
   // GBK_TO_UNICODE[41261] := 16#9B7C;
   // GBK_TO_UNICODE[41262] := 16#F541;
   // GBK_TO_UNICODE[41263] := 16#9B7D;
   // GBK_TO_UNICODE[41264] := 16#F542;
   // GBK_TO_UNICODE[41265] := 16#9B7E;
   // GBK_TO_UNICODE[41266] := 16#F543;
   // GBK_TO_UNICODE[41267] := 16#9B7F;
   // GBK_TO_UNICODE[41268] := 16#F544;
   // GBK_TO_UNICODE[41269] := 16#9B80;
   // GBK_TO_UNICODE[41270] := 16#F545;
   // GBK_TO_UNICODE[41271] := 16#9B81;
   // GBK_TO_UNICODE[41272] := 16#F546;
   // GBK_TO_UNICODE[41273] := 16#9B82;
   // GBK_TO_UNICODE[41274] := 16#F547;
   // GBK_TO_UNICODE[41275] := 16#9B83;
   // GBK_TO_UNICODE[41276] := 16#F548;
   // GBK_TO_UNICODE[41277] := 16#9B84;
   // GBK_TO_UNICODE[41278] := 16#F549;
   // GBK_TO_UNICODE[41279] := 16#9B85;
   // GBK_TO_UNICODE[41280] := 16#F54A;
   // GBK_TO_UNICODE[41281] := 16#9B86;
   // GBK_TO_UNICODE[41282] := 16#F54B;
   // GBK_TO_UNICODE[41283] := 16#9B87;
   // GBK_TO_UNICODE[41284] := 16#F54C;
   // GBK_TO_UNICODE[41285] := 16#9B88;
   // GBK_TO_UNICODE[41286] := 16#F54D;
   // GBK_TO_UNICODE[41287] := 16#9B89;
   // GBK_TO_UNICODE[41288] := 16#F54E;
   // GBK_TO_UNICODE[41289] := 16#9B8A;
   // GBK_TO_UNICODE[41290] := 16#F54F;
   // GBK_TO_UNICODE[41291] := 16#9B8B;
   // GBK_TO_UNICODE[41292] := 16#F550;
   // GBK_TO_UNICODE[41293] := 16#9B8C;
   // GBK_TO_UNICODE[41294] := 16#F551;
   // GBK_TO_UNICODE[41295] := 16#9B8D;
   // GBK_TO_UNICODE[41296] := 16#F552;
   // GBK_TO_UNICODE[41297] := 16#9B8E;
   // GBK_TO_UNICODE[41298] := 16#F553;
   // GBK_TO_UNICODE[41299] := 16#9B8F;
   // GBK_TO_UNICODE[41300] := 16#F554;
   // GBK_TO_UNICODE[41301] := 16#9B90;
   // GBK_TO_UNICODE[41302] := 16#F555;
   // GBK_TO_UNICODE[41303] := 16#9B91;
   // GBK_TO_UNICODE[41304] := 16#F556;
   // GBK_TO_UNICODE[41305] := 16#9B92;
   // GBK_TO_UNICODE[41306] := 16#F557;
   // GBK_TO_UNICODE[41307] := 16#9B93;
   // GBK_TO_UNICODE[41308] := 16#F558;
   // GBK_TO_UNICODE[41309] := 16#9B94;
   // GBK_TO_UNICODE[41310] := 16#F559;
   // GBK_TO_UNICODE[41311] := 16#9B95;
   // GBK_TO_UNICODE[41312] := 16#F55A;
   // GBK_TO_UNICODE[41313] := 16#9B96;
   // GBK_TO_UNICODE[41314] := 16#F55B;
   // GBK_TO_UNICODE[41315] := 16#9B97;
   // GBK_TO_UNICODE[41316] := 16#F55C;
   // GBK_TO_UNICODE[41317] := 16#9B98;
   // GBK_TO_UNICODE[41318] := 16#F55D;
   // GBK_TO_UNICODE[41319] := 16#9B99;
   // GBK_TO_UNICODE[41320] := 16#F55E;
   // GBK_TO_UNICODE[41321] := 16#9B9A;
   // GBK_TO_UNICODE[41322] := 16#F55F;
   // GBK_TO_UNICODE[41323] := 16#9B9B;
   // GBK_TO_UNICODE[41324] := 16#F560;
   // GBK_TO_UNICODE[41325] := 16#9B9C;
   // GBK_TO_UNICODE[41326] := 16#F561;
   // GBK_TO_UNICODE[41327] := 16#9B9D;
   // GBK_TO_UNICODE[41328] := 16#F562;
   // GBK_TO_UNICODE[41329] := 16#9B9E;
   // GBK_TO_UNICODE[41330] := 16#F563;
   // GBK_TO_UNICODE[41331] := 16#9B9F;
   // GBK_TO_UNICODE[41332] := 16#F564;
   // GBK_TO_UNICODE[41333] := 16#9BA0;
   // GBK_TO_UNICODE[41334] := 16#F565;
   // GBK_TO_UNICODE[41335] := 16#9BA1;
   // GBK_TO_UNICODE[41336] := 16#F566;
   // GBK_TO_UNICODE[41337] := 16#9BA2;
   // GBK_TO_UNICODE[41338] := 16#F567;
   // GBK_TO_UNICODE[41339] := 16#9BA3;
   // GBK_TO_UNICODE[41340] := 16#F568;
   // GBK_TO_UNICODE[41341] := 16#9BA4;
   // GBK_TO_UNICODE[41342] := 16#F569;
   // GBK_TO_UNICODE[41343] := 16#9BA5;
   // GBK_TO_UNICODE[41344] := 16#F56A;
   // GBK_TO_UNICODE[41345] := 16#9BA6;
   // GBK_TO_UNICODE[41346] := 16#F56B;
   // GBK_TO_UNICODE[41347] := 16#9BA7;
   // GBK_TO_UNICODE[41348] := 16#F56C;
   // GBK_TO_UNICODE[41349] := 16#9BA8;
   // GBK_TO_UNICODE[41350] := 16#F56D;
   // GBK_TO_UNICODE[41351] := 16#9BA9;
   // GBK_TO_UNICODE[41352] := 16#F56E;
   // GBK_TO_UNICODE[41353] := 16#9BAA;
   // GBK_TO_UNICODE[41354] := 16#F56F;
   // GBK_TO_UNICODE[41355] := 16#9BAB;
   // GBK_TO_UNICODE[41356] := 16#F570;
   // GBK_TO_UNICODE[41357] := 16#9BAC;
   // GBK_TO_UNICODE[41358] := 16#F571;
   // GBK_TO_UNICODE[41359] := 16#9BAD;
   // GBK_TO_UNICODE[41360] := 16#F572;
   // GBK_TO_UNICODE[41361] := 16#9BAE;
   // GBK_TO_UNICODE[41362] := 16#F573;
   // GBK_TO_UNICODE[41363] := 16#9BAF;
   // GBK_TO_UNICODE[41364] := 16#F574;
   // GBK_TO_UNICODE[41365] := 16#9BB0;
   // GBK_TO_UNICODE[41366] := 16#F575;
   // GBK_TO_UNICODE[41367] := 16#9BB1;
   // GBK_TO_UNICODE[41368] := 16#F576;
   // GBK_TO_UNICODE[41369] := 16#9BB2;
   // GBK_TO_UNICODE[41370] := 16#F577;
   // GBK_TO_UNICODE[41371] := 16#9BB3;
   // GBK_TO_UNICODE[41372] := 16#F578;
   // GBK_TO_UNICODE[41373] := 16#9BB4;
   // GBK_TO_UNICODE[41374] := 16#F579;
   // GBK_TO_UNICODE[41375] := 16#9BB5;
   // GBK_TO_UNICODE[41376] := 16#F57A;
   // GBK_TO_UNICODE[41377] := 16#9BB6;
   // GBK_TO_UNICODE[41378] := 16#F57B;
   // GBK_TO_UNICODE[41379] := 16#9BB7;
   // GBK_TO_UNICODE[41380] := 16#F57C;
   // GBK_TO_UNICODE[41381] := 16#9BB8;
   // GBK_TO_UNICODE[41382] := 16#F57D;
   // GBK_TO_UNICODE[41383] := 16#9BB9;
   // GBK_TO_UNICODE[41384] := 16#F57E;
   // GBK_TO_UNICODE[41385] := 16#9BBA;
   // GBK_TO_UNICODE[41386] := 16#F580;
   // GBK_TO_UNICODE[41387] := 16#9BBB;
   // GBK_TO_UNICODE[41388] := 16#F581;
   // GBK_TO_UNICODE[41389] := 16#9BBC;
   // GBK_TO_UNICODE[41390] := 16#F582;
   // GBK_TO_UNICODE[41391] := 16#9BBD;
   // GBK_TO_UNICODE[41392] := 16#F583;
   // GBK_TO_UNICODE[41393] := 16#9BBE;
   // GBK_TO_UNICODE[41394] := 16#F584;
   // GBK_TO_UNICODE[41395] := 16#9BBF;
   // GBK_TO_UNICODE[41396] := 16#F585;
   // GBK_TO_UNICODE[41397] := 16#9BC0;
   // GBK_TO_UNICODE[41398] := 16#F586;
   // GBK_TO_UNICODE[41399] := 16#9BC1;
   // GBK_TO_UNICODE[41400] := 16#F587;
   // GBK_TO_UNICODE[41401] := 16#9BC2;
   // GBK_TO_UNICODE[41402] := 16#F588;
   // GBK_TO_UNICODE[41403] := 16#9BC3;
   // GBK_TO_UNICODE[41404] := 16#F589;
   // GBK_TO_UNICODE[41405] := 16#9BC4;
   // GBK_TO_UNICODE[41406] := 16#F58A;
   // GBK_TO_UNICODE[41407] := 16#9BC5;
   // GBK_TO_UNICODE[41408] := 16#F58B;
   // GBK_TO_UNICODE[41409] := 16#9BC6;
   // GBK_TO_UNICODE[41410] := 16#F58C;
   // GBK_TO_UNICODE[41411] := 16#9BC7;
   // GBK_TO_UNICODE[41412] := 16#F58D;
   // GBK_TO_UNICODE[41413] := 16#9BC8;
   // GBK_TO_UNICODE[41414] := 16#F58E;
   // GBK_TO_UNICODE[41415] := 16#9BC9;
   // GBK_TO_UNICODE[41416] := 16#F58F;
   // GBK_TO_UNICODE[41417] := 16#9BCA;
   // GBK_TO_UNICODE[41418] := 16#F590;
   // GBK_TO_UNICODE[41419] := 16#9BCB;
   // GBK_TO_UNICODE[41420] := 16#F591;
   // GBK_TO_UNICODE[41421] := 16#9BCC;
   // GBK_TO_UNICODE[41422] := 16#F592;
   // GBK_TO_UNICODE[41423] := 16#9BCD;
   // GBK_TO_UNICODE[41424] := 16#F593;
   // GBK_TO_UNICODE[41425] := 16#9BCE;
   // GBK_TO_UNICODE[41426] := 16#F594;
   // GBK_TO_UNICODE[41427] := 16#9BCF;
   // GBK_TO_UNICODE[41428] := 16#F595;
   // GBK_TO_UNICODE[41429] := 16#9BD0;
   // GBK_TO_UNICODE[41430] := 16#F596;
   // GBK_TO_UNICODE[41431] := 16#9BD1;
   // GBK_TO_UNICODE[41432] := 16#F597;
   // GBK_TO_UNICODE[41433] := 16#9BD2;
   // GBK_TO_UNICODE[41434] := 16#F598;
   // GBK_TO_UNICODE[41435] := 16#9BD3;
   // GBK_TO_UNICODE[41436] := 16#F599;
   // GBK_TO_UNICODE[41437] := 16#9BD4;
   // GBK_TO_UNICODE[41438] := 16#F59A;
   // GBK_TO_UNICODE[41439] := 16#9BD5;
   // GBK_TO_UNICODE[41440] := 16#F59B;
   // GBK_TO_UNICODE[41441] := 16#9BD6;
   // GBK_TO_UNICODE[41442] := 16#F59C;
   // GBK_TO_UNICODE[41443] := 16#9BD7;
   // GBK_TO_UNICODE[41444] := 16#F59D;
   // GBK_TO_UNICODE[41445] := 16#9BD8;
   // GBK_TO_UNICODE[41446] := 16#F59E;
   // GBK_TO_UNICODE[41447] := 16#9BD9;
   // GBK_TO_UNICODE[41448] := 16#F59F;
   // GBK_TO_UNICODE[41449] := 16#9BDA;
   // GBK_TO_UNICODE[41450] := 16#F5A0;
   // GBK_TO_UNICODE[41451] := 16#9BDB;
   // GBK_TO_UNICODE[41452] := 16#F5A1;
   // GBK_TO_UNICODE[41453] := 16#9162;
   // GBK_TO_UNICODE[41454] := 16#F5A2;
   // GBK_TO_UNICODE[41455] := 16#9161;
   // GBK_TO_UNICODE[41456] := 16#F5A3;
   // GBK_TO_UNICODE[41457] := 16#9170;
   // GBK_TO_UNICODE[41458] := 16#F5A4;
   // GBK_TO_UNICODE[41459] := 16#9169;
   // GBK_TO_UNICODE[41460] := 16#F5A5;
   // GBK_TO_UNICODE[41461] := 16#916F;
   // GBK_TO_UNICODE[41462] := 16#F5A6;
   // GBK_TO_UNICODE[41463] := 16#917D;
   // GBK_TO_UNICODE[41464] := 16#F5A7;
   // GBK_TO_UNICODE[41465] := 16#917E;
   // GBK_TO_UNICODE[41466] := 16#F5A8;
   // GBK_TO_UNICODE[41467] := 16#9172;
   // GBK_TO_UNICODE[41468] := 16#F5A9;
   // GBK_TO_UNICODE[41469] := 16#9174;
   // GBK_TO_UNICODE[41470] := 16#F5AA;
   // GBK_TO_UNICODE[41471] := 16#9179;
   // GBK_TO_UNICODE[41472] := 16#F5AB;
   // GBK_TO_UNICODE[41473] := 16#918C;
   // GBK_TO_UNICODE[41474] := 16#F5AC;
   // GBK_TO_UNICODE[41475] := 16#9185;
   // GBK_TO_UNICODE[41476] := 16#F5AD;
   // GBK_TO_UNICODE[41477] := 16#9190;
   // GBK_TO_UNICODE[41478] := 16#F5AE;
   // GBK_TO_UNICODE[41479] := 16#918D;
   // GBK_TO_UNICODE[41480] := 16#F5AF;
   // GBK_TO_UNICODE[41481] := 16#9191;
   // GBK_TO_UNICODE[41482] := 16#F5B0;
   // GBK_TO_UNICODE[41483] := 16#91A2;
   // GBK_TO_UNICODE[41484] := 16#F5B1;
   // GBK_TO_UNICODE[41485] := 16#91A3;
   // GBK_TO_UNICODE[41486] := 16#F5B2;
   // GBK_TO_UNICODE[41487] := 16#91AA;
   // GBK_TO_UNICODE[41488] := 16#F5B3;
   // GBK_TO_UNICODE[41489] := 16#91AD;
   // GBK_TO_UNICODE[41490] := 16#F5B4;
   // GBK_TO_UNICODE[41491] := 16#91AE;
   // GBK_TO_UNICODE[41492] := 16#F5B5;
   // GBK_TO_UNICODE[41493] := 16#91AF;
   // GBK_TO_UNICODE[41494] := 16#F5B6;
   // GBK_TO_UNICODE[41495] := 16#91B5;
   // GBK_TO_UNICODE[41496] := 16#F5B7;
   // GBK_TO_UNICODE[41497] := 16#91B4;
   // GBK_TO_UNICODE[41498] := 16#F5B8;
   // GBK_TO_UNICODE[41499] := 16#91BA;
   // GBK_TO_UNICODE[41500] := 16#F5B9;
   // GBK_TO_UNICODE[41501] := 16#8C55;
   // GBK_TO_UNICODE[41502] := 16#F5BA;
   // GBK_TO_UNICODE[41503] := 16#9E7E;
   // GBK_TO_UNICODE[41504] := 16#F5BB;
   // GBK_TO_UNICODE[41505] := 16#8DB8;
   // GBK_TO_UNICODE[41506] := 16#F5BC;
   // GBK_TO_UNICODE[41507] := 16#8DEB;
   // GBK_TO_UNICODE[41508] := 16#F5BD;
   // GBK_TO_UNICODE[41509] := 16#8E05;
   // GBK_TO_UNICODE[41510] := 16#F5BE;
   // GBK_TO_UNICODE[41511] := 16#8E59;
   // GBK_TO_UNICODE[41512] := 16#F5BF;
   // GBK_TO_UNICODE[41513] := 16#8E69;
   // GBK_TO_UNICODE[41514] := 16#F5C0;
   // GBK_TO_UNICODE[41515] := 16#8DB5;
   // GBK_TO_UNICODE[41516] := 16#F5C1;
   // GBK_TO_UNICODE[41517] := 16#8DBF;
   // GBK_TO_UNICODE[41518] := 16#F5C2;
   // GBK_TO_UNICODE[41519] := 16#8DBC;
   // GBK_TO_UNICODE[41520] := 16#F5C3;
   // GBK_TO_UNICODE[41521] := 16#8DBA;
   // GBK_TO_UNICODE[41522] := 16#F5C4;
   // GBK_TO_UNICODE[41523] := 16#8DC4;
   // GBK_TO_UNICODE[41524] := 16#F5C5;
   // GBK_TO_UNICODE[41525] := 16#8DD6;
   // GBK_TO_UNICODE[41526] := 16#F5C6;
   // GBK_TO_UNICODE[41527] := 16#8DD7;
   // GBK_TO_UNICODE[41528] := 16#F5C7;
   // GBK_TO_UNICODE[41529] := 16#8DDA;
   // GBK_TO_UNICODE[41530] := 16#F5C8;
   // GBK_TO_UNICODE[41531] := 16#8DDE;
   // GBK_TO_UNICODE[41532] := 16#F5C9;
   // GBK_TO_UNICODE[41533] := 16#8DCE;
   // GBK_TO_UNICODE[41534] := 16#F5CA;
   // GBK_TO_UNICODE[41535] := 16#8DCF;
   // GBK_TO_UNICODE[41536] := 16#F5CB;
   // GBK_TO_UNICODE[41537] := 16#8DDB;
   // GBK_TO_UNICODE[41538] := 16#F5CC;
   // GBK_TO_UNICODE[41539] := 16#8DC6;
   // GBK_TO_UNICODE[41540] := 16#F5CD;
   // GBK_TO_UNICODE[41541] := 16#8DEC;
   // GBK_TO_UNICODE[41542] := 16#F5CE;
   // GBK_TO_UNICODE[41543] := 16#8DF7;
   // GBK_TO_UNICODE[41544] := 16#F5CF;
   // GBK_TO_UNICODE[41545] := 16#8DF8;
   // GBK_TO_UNICODE[41546] := 16#F5D0;
   // GBK_TO_UNICODE[41547] := 16#8DE3;
   // GBK_TO_UNICODE[41548] := 16#F5D1;
   // GBK_TO_UNICODE[41549] := 16#8DF9;
   // GBK_TO_UNICODE[41550] := 16#F5D2;
   // GBK_TO_UNICODE[41551] := 16#8DFB;
   // GBK_TO_UNICODE[41552] := 16#F5D3;
   // GBK_TO_UNICODE[41553] := 16#8DE4;
   // GBK_TO_UNICODE[41554] := 16#F5D4;
   // GBK_TO_UNICODE[41555] := 16#8E09;
   // GBK_TO_UNICODE[41556] := 16#F5D5;
   // GBK_TO_UNICODE[41557] := 16#8DFD;
   // GBK_TO_UNICODE[41558] := 16#F5D6;
   // GBK_TO_UNICODE[41559] := 16#8E14;
   // GBK_TO_UNICODE[41560] := 16#F5D7;
   // GBK_TO_UNICODE[41561] := 16#8E1D;
   // GBK_TO_UNICODE[41562] := 16#F5D8;
   // GBK_TO_UNICODE[41563] := 16#8E1F;
   // GBK_TO_UNICODE[41564] := 16#F5D9;
   // GBK_TO_UNICODE[41565] := 16#8E2C;
   // GBK_TO_UNICODE[41566] := 16#F5DA;
   // GBK_TO_UNICODE[41567] := 16#8E2E;
   // GBK_TO_UNICODE[41568] := 16#F5DB;
   // GBK_TO_UNICODE[41569] := 16#8E23;
   // GBK_TO_UNICODE[41570] := 16#F5DC;
   // GBK_TO_UNICODE[41571] := 16#8E2F;
   // GBK_TO_UNICODE[41572] := 16#F5DD;
   // GBK_TO_UNICODE[41573] := 16#8E3A;
   // GBK_TO_UNICODE[41574] := 16#F5DE;
   // GBK_TO_UNICODE[41575] := 16#8E40;
   // GBK_TO_UNICODE[41576] := 16#F5DF;
   // GBK_TO_UNICODE[41577] := 16#8E39;
   // GBK_TO_UNICODE[41578] := 16#F5E0;
   // GBK_TO_UNICODE[41579] := 16#8E35;
   // GBK_TO_UNICODE[41580] := 16#F5E1;
   // GBK_TO_UNICODE[41581] := 16#8E3D;
   // GBK_TO_UNICODE[41582] := 16#F5E2;
   // GBK_TO_UNICODE[41583] := 16#8E31;
   // GBK_TO_UNICODE[41584] := 16#F5E3;
   // GBK_TO_UNICODE[41585] := 16#8E49;
   // GBK_TO_UNICODE[41586] := 16#F5E4;
   // GBK_TO_UNICODE[41587] := 16#8E41;
   // GBK_TO_UNICODE[41588] := 16#F5E5;
   // GBK_TO_UNICODE[41589] := 16#8E42;
   // GBK_TO_UNICODE[41590] := 16#F5E6;
   // GBK_TO_UNICODE[41591] := 16#8E51;
   // GBK_TO_UNICODE[41592] := 16#F5E7;
   // GBK_TO_UNICODE[41593] := 16#8E52;
   // GBK_TO_UNICODE[41594] := 16#F5E8;
   // GBK_TO_UNICODE[41595] := 16#8E4A;
   // GBK_TO_UNICODE[41596] := 16#F5E9;
   // GBK_TO_UNICODE[41597] := 16#8E70;
   // GBK_TO_UNICODE[41598] := 16#F5EA;
   // GBK_TO_UNICODE[41599] := 16#8E76;
   // GBK_TO_UNICODE[41600] := 16#F5EB;
   // GBK_TO_UNICODE[41601] := 16#8E7C;
   // GBK_TO_UNICODE[41602] := 16#F5EC;
   // GBK_TO_UNICODE[41603] := 16#8E6F;
   // GBK_TO_UNICODE[41604] := 16#F5ED;
   // GBK_TO_UNICODE[41605] := 16#8E74;
   // GBK_TO_UNICODE[41606] := 16#F5EE;
   // GBK_TO_UNICODE[41607] := 16#8E85;
   // GBK_TO_UNICODE[41608] := 16#F5EF;
   // GBK_TO_UNICODE[41609] := 16#8E8F;
   // GBK_TO_UNICODE[41610] := 16#F5F0;
   // GBK_TO_UNICODE[41611] := 16#8E94;
   // GBK_TO_UNICODE[41612] := 16#F5F1;
   // GBK_TO_UNICODE[41613] := 16#8E90;
   // GBK_TO_UNICODE[41614] := 16#F5F2;
   // GBK_TO_UNICODE[41615] := 16#8E9C;
   // GBK_TO_UNICODE[41616] := 16#F5F3;
   // GBK_TO_UNICODE[41617] := 16#8E9E;
   // GBK_TO_UNICODE[41618] := 16#F5F4;
   // GBK_TO_UNICODE[41619] := 16#8C78;
   // GBK_TO_UNICODE[41620] := 16#F5F5;
   // GBK_TO_UNICODE[41621] := 16#8C82;
   // GBK_TO_UNICODE[41622] := 16#F5F6;
   // GBK_TO_UNICODE[41623] := 16#8C8A;
   // GBK_TO_UNICODE[41624] := 16#F5F7;
   // GBK_TO_UNICODE[41625] := 16#8C85;
   // GBK_TO_UNICODE[41626] := 16#F5F8;
   // GBK_TO_UNICODE[41627] := 16#8C98;
   // GBK_TO_UNICODE[41628] := 16#F5F9;
   // GBK_TO_UNICODE[41629] := 16#8C94;
   // GBK_TO_UNICODE[41630] := 16#F5FA;
   // GBK_TO_UNICODE[41631] := 16#659B;
   // GBK_TO_UNICODE[41632] := 16#F5FB;
   // GBK_TO_UNICODE[41633] := 16#89D6;
   // GBK_TO_UNICODE[41634] := 16#F5FC;
   // GBK_TO_UNICODE[41635] := 16#89DE;
   // GBK_TO_UNICODE[41636] := 16#F5FD;
   // GBK_TO_UNICODE[41637] := 16#89DA;
   // GBK_TO_UNICODE[41638] := 16#F5FE;
   // GBK_TO_UNICODE[41639] := 16#89DC;
   // GBK_TO_UNICODE[41640] := 16#F640;
   // GBK_TO_UNICODE[41641] := 16#9BDC;
   // GBK_TO_UNICODE[41642] := 16#F641;
   // GBK_TO_UNICODE[41643] := 16#9BDD;
   // GBK_TO_UNICODE[41644] := 16#F642;
   // GBK_TO_UNICODE[41645] := 16#9BDE;
   // GBK_TO_UNICODE[41646] := 16#F643;
   // GBK_TO_UNICODE[41647] := 16#9BDF;
   // GBK_TO_UNICODE[41648] := 16#F644;
   // GBK_TO_UNICODE[41649] := 16#9BE0;
   // GBK_TO_UNICODE[41650] := 16#F645;
   // GBK_TO_UNICODE[41651] := 16#9BE1;
   // GBK_TO_UNICODE[41652] := 16#F646;
   // GBK_TO_UNICODE[41653] := 16#9BE2;
   // GBK_TO_UNICODE[41654] := 16#F647;
   // GBK_TO_UNICODE[41655] := 16#9BE3;
   // GBK_TO_UNICODE[41656] := 16#F648;
   // GBK_TO_UNICODE[41657] := 16#9BE4;
   // GBK_TO_UNICODE[41658] := 16#F649;
   // GBK_TO_UNICODE[41659] := 16#9BE5;
   // GBK_TO_UNICODE[41660] := 16#F64A;
   // GBK_TO_UNICODE[41661] := 16#9BE6;
   // GBK_TO_UNICODE[41662] := 16#F64B;
   // GBK_TO_UNICODE[41663] := 16#9BE7;
   // GBK_TO_UNICODE[41664] := 16#F64C;
   // GBK_TO_UNICODE[41665] := 16#9BE8;
   // GBK_TO_UNICODE[41666] := 16#F64D;
   // GBK_TO_UNICODE[41667] := 16#9BE9;
   // GBK_TO_UNICODE[41668] := 16#F64E;
   // GBK_TO_UNICODE[41669] := 16#9BEA;
   // GBK_TO_UNICODE[41670] := 16#F64F;
   // GBK_TO_UNICODE[41671] := 16#9BEB;
   // GBK_TO_UNICODE[41672] := 16#F650;
   // GBK_TO_UNICODE[41673] := 16#9BEC;
   // GBK_TO_UNICODE[41674] := 16#F651;
   // GBK_TO_UNICODE[41675] := 16#9BED;
   // GBK_TO_UNICODE[41676] := 16#F652;
   // GBK_TO_UNICODE[41677] := 16#9BEE;
   // GBK_TO_UNICODE[41678] := 16#F653;
   // GBK_TO_UNICODE[41679] := 16#9BEF;
   // GBK_TO_UNICODE[41680] := 16#F654;
   // GBK_TO_UNICODE[41681] := 16#9BF0;
   // GBK_TO_UNICODE[41682] := 16#F655;
   // GBK_TO_UNICODE[41683] := 16#9BF1;
   // GBK_TO_UNICODE[41684] := 16#F656;
   // GBK_TO_UNICODE[41685] := 16#9BF2;
   // GBK_TO_UNICODE[41686] := 16#F657;
   // GBK_TO_UNICODE[41687] := 16#9BF3;
   // GBK_TO_UNICODE[41688] := 16#F658;
   // GBK_TO_UNICODE[41689] := 16#9BF4;
   // GBK_TO_UNICODE[41690] := 16#F659;
   // GBK_TO_UNICODE[41691] := 16#9BF5;
   // GBK_TO_UNICODE[41692] := 16#F65A;
   // GBK_TO_UNICODE[41693] := 16#9BF6;
   // GBK_TO_UNICODE[41694] := 16#F65B;
   // GBK_TO_UNICODE[41695] := 16#9BF7;
   // GBK_TO_UNICODE[41696] := 16#F65C;
   // GBK_TO_UNICODE[41697] := 16#9BF8;
   // GBK_TO_UNICODE[41698] := 16#F65D;
   // GBK_TO_UNICODE[41699] := 16#9BF9;
   // GBK_TO_UNICODE[41700] := 16#F65E;
   // GBK_TO_UNICODE[41701] := 16#9BFA;
   // GBK_TO_UNICODE[41702] := 16#F65F;
   // GBK_TO_UNICODE[41703] := 16#9BFB;
   // GBK_TO_UNICODE[41704] := 16#F660;
   // GBK_TO_UNICODE[41705] := 16#9BFC;
   // GBK_TO_UNICODE[41706] := 16#F661;
   // GBK_TO_UNICODE[41707] := 16#9BFD;
   // GBK_TO_UNICODE[41708] := 16#F662;
   // GBK_TO_UNICODE[41709] := 16#9BFE;
   // GBK_TO_UNICODE[41710] := 16#F663;
   // GBK_TO_UNICODE[41711] := 16#9BFF;
   // GBK_TO_UNICODE[41712] := 16#F664;
   // GBK_TO_UNICODE[41713] := 16#9C00;
   // GBK_TO_UNICODE[41714] := 16#F665;
   // GBK_TO_UNICODE[41715] := 16#9C01;
   // GBK_TO_UNICODE[41716] := 16#F666;
   // GBK_TO_UNICODE[41717] := 16#9C02;
   // GBK_TO_UNICODE[41718] := 16#F667;
   // GBK_TO_UNICODE[41719] := 16#9C03;
   // GBK_TO_UNICODE[41720] := 16#F668;
   // GBK_TO_UNICODE[41721] := 16#9C04;
   // GBK_TO_UNICODE[41722] := 16#F669;
   // GBK_TO_UNICODE[41723] := 16#9C05;
   // GBK_TO_UNICODE[41724] := 16#F66A;
   // GBK_TO_UNICODE[41725] := 16#9C06;
   // GBK_TO_UNICODE[41726] := 16#F66B;
   // GBK_TO_UNICODE[41727] := 16#9C07;
   // GBK_TO_UNICODE[41728] := 16#F66C;
   // GBK_TO_UNICODE[41729] := 16#9C08;
   // GBK_TO_UNICODE[41730] := 16#F66D;
   // GBK_TO_UNICODE[41731] := 16#9C09;
   // GBK_TO_UNICODE[41732] := 16#F66E;
   // GBK_TO_UNICODE[41733] := 16#9C0A;
   // GBK_TO_UNICODE[41734] := 16#F66F;
   // GBK_TO_UNICODE[41735] := 16#9C0B;
   // GBK_TO_UNICODE[41736] := 16#F670;
   // GBK_TO_UNICODE[41737] := 16#9C0C;
   // GBK_TO_UNICODE[41738] := 16#F671;
   // GBK_TO_UNICODE[41739] := 16#9C0D;
   // GBK_TO_UNICODE[41740] := 16#F672;
   // GBK_TO_UNICODE[41741] := 16#9C0E;
   // GBK_TO_UNICODE[41742] := 16#F673;
   // GBK_TO_UNICODE[41743] := 16#9C0F;
   // GBK_TO_UNICODE[41744] := 16#F674;
   // GBK_TO_UNICODE[41745] := 16#9C10;
   // GBK_TO_UNICODE[41746] := 16#F675;
   // GBK_TO_UNICODE[41747] := 16#9C11;
   // GBK_TO_UNICODE[41748] := 16#F676;
   // GBK_TO_UNICODE[41749] := 16#9C12;
   // GBK_TO_UNICODE[41750] := 16#F677;
   // GBK_TO_UNICODE[41751] := 16#9C13;
   // GBK_TO_UNICODE[41752] := 16#F678;
   // GBK_TO_UNICODE[41753] := 16#9C14;
   // GBK_TO_UNICODE[41754] := 16#F679;
   // GBK_TO_UNICODE[41755] := 16#9C15;
   // GBK_TO_UNICODE[41756] := 16#F67A;
   // GBK_TO_UNICODE[41757] := 16#9C16;
   // GBK_TO_UNICODE[41758] := 16#F67B;
   // GBK_TO_UNICODE[41759] := 16#9C17;
   // GBK_TO_UNICODE[41760] := 16#F67C;
   // GBK_TO_UNICODE[41761] := 16#9C18;
   // GBK_TO_UNICODE[41762] := 16#F67D;
   // GBK_TO_UNICODE[41763] := 16#9C19;
   // GBK_TO_UNICODE[41764] := 16#F67E;
   // GBK_TO_UNICODE[41765] := 16#9C1A;
   // GBK_TO_UNICODE[41766] := 16#F680;
   // GBK_TO_UNICODE[41767] := 16#9C1B;
   // GBK_TO_UNICODE[41768] := 16#F681;
   // GBK_TO_UNICODE[41769] := 16#9C1C;
   // GBK_TO_UNICODE[41770] := 16#F682;
   // GBK_TO_UNICODE[41771] := 16#9C1D;
   // GBK_TO_UNICODE[41772] := 16#F683;
   // GBK_TO_UNICODE[41773] := 16#9C1E;
   // GBK_TO_UNICODE[41774] := 16#F684;
   // GBK_TO_UNICODE[41775] := 16#9C1F;
   // GBK_TO_UNICODE[41776] := 16#F685;
   // GBK_TO_UNICODE[41777] := 16#9C20;
   // GBK_TO_UNICODE[41778] := 16#F686;
   // GBK_TO_UNICODE[41779] := 16#9C21;
   // GBK_TO_UNICODE[41780] := 16#F687;
   // GBK_TO_UNICODE[41781] := 16#9C22;
   // GBK_TO_UNICODE[41782] := 16#F688;
   // GBK_TO_UNICODE[41783] := 16#9C23;
   // GBK_TO_UNICODE[41784] := 16#F689;
   // GBK_TO_UNICODE[41785] := 16#9C24;
   // GBK_TO_UNICODE[41786] := 16#F68A;
   // GBK_TO_UNICODE[41787] := 16#9C25;
   // GBK_TO_UNICODE[41788] := 16#F68B;
   // GBK_TO_UNICODE[41789] := 16#9C26;
   // GBK_TO_UNICODE[41790] := 16#F68C;
   // GBK_TO_UNICODE[41791] := 16#9C27;
   // GBK_TO_UNICODE[41792] := 16#F68D;
   // GBK_TO_UNICODE[41793] := 16#9C28;
   // GBK_TO_UNICODE[41794] := 16#F68E;
   // GBK_TO_UNICODE[41795] := 16#9C29;
   // GBK_TO_UNICODE[41796] := 16#F68F;
   // GBK_TO_UNICODE[41797] := 16#9C2A;
   // GBK_TO_UNICODE[41798] := 16#F690;
   // GBK_TO_UNICODE[41799] := 16#9C2B;
   // GBK_TO_UNICODE[41800] := 16#F691;
   // GBK_TO_UNICODE[41801] := 16#9C2C;
   // GBK_TO_UNICODE[41802] := 16#F692;
   // GBK_TO_UNICODE[41803] := 16#9C2D;
   // GBK_TO_UNICODE[41804] := 16#F693;
   // GBK_TO_UNICODE[41805] := 16#9C2E;
   // GBK_TO_UNICODE[41806] := 16#F694;
   // GBK_TO_UNICODE[41807] := 16#9C2F;
   // GBK_TO_UNICODE[41808] := 16#F695;
   // GBK_TO_UNICODE[41809] := 16#9C30;
   // GBK_TO_UNICODE[41810] := 16#F696;
   // GBK_TO_UNICODE[41811] := 16#9C31;
   // GBK_TO_UNICODE[41812] := 16#F697;
   // GBK_TO_UNICODE[41813] := 16#9C32;
   // GBK_TO_UNICODE[41814] := 16#F698;
   // GBK_TO_UNICODE[41815] := 16#9C33;
   // GBK_TO_UNICODE[41816] := 16#F699;
   // GBK_TO_UNICODE[41817] := 16#9C34;
   // GBK_TO_UNICODE[41818] := 16#F69A;
   // GBK_TO_UNICODE[41819] := 16#9C35;
   // GBK_TO_UNICODE[41820] := 16#F69B;
   // GBK_TO_UNICODE[41821] := 16#9C36;
   // GBK_TO_UNICODE[41822] := 16#F69C;
   // GBK_TO_UNICODE[41823] := 16#9C37;
   // GBK_TO_UNICODE[41824] := 16#F69D;
   // GBK_TO_UNICODE[41825] := 16#9C38;
   // GBK_TO_UNICODE[41826] := 16#F69E;
   // GBK_TO_UNICODE[41827] := 16#9C39;
   // GBK_TO_UNICODE[41828] := 16#F69F;
   // GBK_TO_UNICODE[41829] := 16#9C3A;
   // GBK_TO_UNICODE[41830] := 16#F6A0;
   // GBK_TO_UNICODE[41831] := 16#9C3B;
   // GBK_TO_UNICODE[41832] := 16#F6A1;
   // GBK_TO_UNICODE[41833] := 16#89E5;
   // GBK_TO_UNICODE[41834] := 16#F6A2;
   // GBK_TO_UNICODE[41835] := 16#89EB;
   // GBK_TO_UNICODE[41836] := 16#F6A3;
   // GBK_TO_UNICODE[41837] := 16#89EF;
   // GBK_TO_UNICODE[41838] := 16#F6A4;
   // GBK_TO_UNICODE[41839] := 16#8A3E;
   // GBK_TO_UNICODE[41840] := 16#F6A5;
   // GBK_TO_UNICODE[41841] := 16#8B26;
   // GBK_TO_UNICODE[41842] := 16#F6A6;
   // GBK_TO_UNICODE[41843] := 16#9753;
   // GBK_TO_UNICODE[41844] := 16#F6A7;
   // GBK_TO_UNICODE[41845] := 16#96E9;
   // GBK_TO_UNICODE[41846] := 16#F6A8;
   // GBK_TO_UNICODE[41847] := 16#96F3;
   // GBK_TO_UNICODE[41848] := 16#F6A9;
   // GBK_TO_UNICODE[41849] := 16#96EF;
   // GBK_TO_UNICODE[41850] := 16#F6AA;
   // GBK_TO_UNICODE[41851] := 16#9706;
   // GBK_TO_UNICODE[41852] := 16#F6AB;
   // GBK_TO_UNICODE[41853] := 16#9701;
   // GBK_TO_UNICODE[41854] := 16#F6AC;
   // GBK_TO_UNICODE[41855] := 16#9708;
   // GBK_TO_UNICODE[41856] := 16#F6AD;
   // GBK_TO_UNICODE[41857] := 16#970F;
   // GBK_TO_UNICODE[41858] := 16#F6AE;
   // GBK_TO_UNICODE[41859] := 16#970E;
   // GBK_TO_UNICODE[41860] := 16#F6AF;
   // GBK_TO_UNICODE[41861] := 16#972A;
   // GBK_TO_UNICODE[41862] := 16#F6B0;
   // GBK_TO_UNICODE[41863] := 16#972D;
   // GBK_TO_UNICODE[41864] := 16#F6B1;
   // GBK_TO_UNICODE[41865] := 16#9730;
   // GBK_TO_UNICODE[41866] := 16#F6B2;
   // GBK_TO_UNICODE[41867] := 16#973E;
   // GBK_TO_UNICODE[41868] := 16#F6B3;
   // GBK_TO_UNICODE[41869] := 16#9F80;
   // GBK_TO_UNICODE[41870] := 16#F6B4;
   // GBK_TO_UNICODE[41871] := 16#9F83;
   // GBK_TO_UNICODE[41872] := 16#F6B5;
   // GBK_TO_UNICODE[41873] := 16#9F85;
   // GBK_TO_UNICODE[41874] := 16#F6B6;
   // GBK_TO_UNICODE[41875] := 16#9F86;
   // GBK_TO_UNICODE[41876] := 16#F6B7;
   // GBK_TO_UNICODE[41877] := 16#9F87;
   // GBK_TO_UNICODE[41878] := 16#F6B8;
   // GBK_TO_UNICODE[41879] := 16#9F88;
   // GBK_TO_UNICODE[41880] := 16#F6B9;
   // GBK_TO_UNICODE[41881] := 16#9F89;
   // GBK_TO_UNICODE[41882] := 16#F6BA;
   // GBK_TO_UNICODE[41883] := 16#9F8A;
   // GBK_TO_UNICODE[41884] := 16#F6BB;
   // GBK_TO_UNICODE[41885] := 16#9F8C;
   // GBK_TO_UNICODE[41886] := 16#F6BC;
   // GBK_TO_UNICODE[41887] := 16#9EFE;
   // GBK_TO_UNICODE[41888] := 16#F6BD;
   // GBK_TO_UNICODE[41889] := 16#9F0B;
   // GBK_TO_UNICODE[41890] := 16#F6BE;
   // GBK_TO_UNICODE[41891] := 16#9F0D;
   // GBK_TO_UNICODE[41892] := 16#F6BF;
   // GBK_TO_UNICODE[41893] := 16#96B9;
   // GBK_TO_UNICODE[41894] := 16#F6C0;
   // GBK_TO_UNICODE[41895] := 16#96BC;
   // GBK_TO_UNICODE[41896] := 16#F6C1;
   // GBK_TO_UNICODE[41897] := 16#96BD;
   // GBK_TO_UNICODE[41898] := 16#F6C2;
   // GBK_TO_UNICODE[41899] := 16#96CE;
   // GBK_TO_UNICODE[41900] := 16#F6C3;
   // GBK_TO_UNICODE[41901] := 16#96D2;
   // GBK_TO_UNICODE[41902] := 16#F6C4;
   // GBK_TO_UNICODE[41903] := 16#77BF;
   // GBK_TO_UNICODE[41904] := 16#F6C5;
   // GBK_TO_UNICODE[41905] := 16#96E0;
   // GBK_TO_UNICODE[41906] := 16#F6C6;
   // GBK_TO_UNICODE[41907] := 16#928E;
   // GBK_TO_UNICODE[41908] := 16#F6C7;
   // GBK_TO_UNICODE[41909] := 16#92AE;
   // GBK_TO_UNICODE[41910] := 16#F6C8;
   // GBK_TO_UNICODE[41911] := 16#92C8;
   // GBK_TO_UNICODE[41912] := 16#F6C9;
   // GBK_TO_UNICODE[41913] := 16#933E;
   // GBK_TO_UNICODE[41914] := 16#F6CA;
   // GBK_TO_UNICODE[41915] := 16#936A;
   // GBK_TO_UNICODE[41916] := 16#F6CB;
   // GBK_TO_UNICODE[41917] := 16#93CA;
   // GBK_TO_UNICODE[41918] := 16#F6CC;
   // GBK_TO_UNICODE[41919] := 16#938F;
   // GBK_TO_UNICODE[41920] := 16#F6CD;
   // GBK_TO_UNICODE[41921] := 16#943E;
   // GBK_TO_UNICODE[41922] := 16#F6CE;
   // GBK_TO_UNICODE[41923] := 16#946B;
   // GBK_TO_UNICODE[41924] := 16#F6CF;
   // GBK_TO_UNICODE[41925] := 16#9C7F;
   // GBK_TO_UNICODE[41926] := 16#F6D0;
   // GBK_TO_UNICODE[41927] := 16#9C82;
   // GBK_TO_UNICODE[41928] := 16#F6D1;
   // GBK_TO_UNICODE[41929] := 16#9C85;
   // GBK_TO_UNICODE[41930] := 16#F6D2;
   // GBK_TO_UNICODE[41931] := 16#9C86;
   // GBK_TO_UNICODE[41932] := 16#F6D3;
   // GBK_TO_UNICODE[41933] := 16#9C87;
   // GBK_TO_UNICODE[41934] := 16#F6D4;
   // GBK_TO_UNICODE[41935] := 16#9C88;
   // GBK_TO_UNICODE[41936] := 16#F6D5;
   // GBK_TO_UNICODE[41937] := 16#7A23;
   // GBK_TO_UNICODE[41938] := 16#F6D6;
   // GBK_TO_UNICODE[41939] := 16#9C8B;
   // GBK_TO_UNICODE[41940] := 16#F6D7;
   // GBK_TO_UNICODE[41941] := 16#9C8E;
   // GBK_TO_UNICODE[41942] := 16#F6D8;
   // GBK_TO_UNICODE[41943] := 16#9C90;
   // GBK_TO_UNICODE[41944] := 16#F6D9;
   // GBK_TO_UNICODE[41945] := 16#9C91;
   // GBK_TO_UNICODE[41946] := 16#F6DA;
   // GBK_TO_UNICODE[41947] := 16#9C92;
   // GBK_TO_UNICODE[41948] := 16#F6DB;
   // GBK_TO_UNICODE[41949] := 16#9C94;
   // GBK_TO_UNICODE[41950] := 16#F6DC;
   // GBK_TO_UNICODE[41951] := 16#9C95;
   // GBK_TO_UNICODE[41952] := 16#F6DD;
   // GBK_TO_UNICODE[41953] := 16#9C9A;
   // GBK_TO_UNICODE[41954] := 16#F6DE;
   // GBK_TO_UNICODE[41955] := 16#9C9B;
   // GBK_TO_UNICODE[41956] := 16#F6DF;
   // GBK_TO_UNICODE[41957] := 16#9C9E;
   // GBK_TO_UNICODE[41958] := 16#F6E0;
   // GBK_TO_UNICODE[41959] := 16#9C9F;
   // GBK_TO_UNICODE[41960] := 16#F6E1;
   // GBK_TO_UNICODE[41961] := 16#9CA0;
   // GBK_TO_UNICODE[41962] := 16#F6E2;
   // GBK_TO_UNICODE[41963] := 16#9CA1;
   // GBK_TO_UNICODE[41964] := 16#F6E3;
   // GBK_TO_UNICODE[41965] := 16#9CA2;
   // GBK_TO_UNICODE[41966] := 16#F6E4;
   // GBK_TO_UNICODE[41967] := 16#9CA3;
   // GBK_TO_UNICODE[41968] := 16#F6E5;
   // GBK_TO_UNICODE[41969] := 16#9CA5;
   // GBK_TO_UNICODE[41970] := 16#F6E6;
   // GBK_TO_UNICODE[41971] := 16#9CA6;
   // GBK_TO_UNICODE[41972] := 16#F6E7;
   // GBK_TO_UNICODE[41973] := 16#9CA7;
   // GBK_TO_UNICODE[41974] := 16#F6E8;
   // GBK_TO_UNICODE[41975] := 16#9CA8;
   // GBK_TO_UNICODE[41976] := 16#F6E9;
   // GBK_TO_UNICODE[41977] := 16#9CA9;
   // GBK_TO_UNICODE[41978] := 16#F6EA;
   // GBK_TO_UNICODE[41979] := 16#9CAB;
   // GBK_TO_UNICODE[41980] := 16#F6EB;
   // GBK_TO_UNICODE[41981] := 16#9CAD;
   // GBK_TO_UNICODE[41982] := 16#F6EC;
   // GBK_TO_UNICODE[41983] := 16#9CAE;
   // GBK_TO_UNICODE[41984] := 16#F6ED;
   // GBK_TO_UNICODE[41985] := 16#9CB0;
   // GBK_TO_UNICODE[41986] := 16#F6EE;
   // GBK_TO_UNICODE[41987] := 16#9CB1;
   // GBK_TO_UNICODE[41988] := 16#F6EF;
   // GBK_TO_UNICODE[41989] := 16#9CB2;
   // GBK_TO_UNICODE[41990] := 16#F6F0;
   // GBK_TO_UNICODE[41991] := 16#9CB3;
   // GBK_TO_UNICODE[41992] := 16#F6F1;
   // GBK_TO_UNICODE[41993] := 16#9CB4;
   // GBK_TO_UNICODE[41994] := 16#F6F2;
   // GBK_TO_UNICODE[41995] := 16#9CB5;
   // GBK_TO_UNICODE[41996] := 16#F6F3;
   // GBK_TO_UNICODE[41997] := 16#9CB6;
   // GBK_TO_UNICODE[41998] := 16#F6F4;
   // GBK_TO_UNICODE[41999] := 16#9CB7;
   // GBK_TO_UNICODE[42000] := 16#F6F5;
   // GBK_TO_UNICODE[42001] := 16#9CBA;
   // GBK_TO_UNICODE[42002] := 16#F6F6;
   // GBK_TO_UNICODE[42003] := 16#9CBB;
   // GBK_TO_UNICODE[42004] := 16#F6F7;
   // GBK_TO_UNICODE[42005] := 16#9CBC;
   // GBK_TO_UNICODE[42006] := 16#F6F8;
   // GBK_TO_UNICODE[42007] := 16#9CBD;
   // GBK_TO_UNICODE[42008] := 16#F6F9;
   // GBK_TO_UNICODE[42009] := 16#9CC4;
   // GBK_TO_UNICODE[42010] := 16#F6FA;
   // GBK_TO_UNICODE[42011] := 16#9CC5;
   // GBK_TO_UNICODE[42012] := 16#F6FB;
   // GBK_TO_UNICODE[42013] := 16#9CC6;
   // GBK_TO_UNICODE[42014] := 16#F6FC;
   // GBK_TO_UNICODE[42015] := 16#9CC7;
   // GBK_TO_UNICODE[42016] := 16#F6FD;
   // GBK_TO_UNICODE[42017] := 16#9CCA;
   // GBK_TO_UNICODE[42018] := 16#F6FE;
   // GBK_TO_UNICODE[42019] := 16#9CCB;
   // GBK_TO_UNICODE[42020] := 16#F740;
   // GBK_TO_UNICODE[42021] := 16#9C3C;
   // GBK_TO_UNICODE[42022] := 16#F741;
   // GBK_TO_UNICODE[42023] := 16#9C3D;
   // GBK_TO_UNICODE[42024] := 16#F742;
   // GBK_TO_UNICODE[42025] := 16#9C3E;
   // GBK_TO_UNICODE[42026] := 16#F743;
   // GBK_TO_UNICODE[42027] := 16#9C3F;
   // GBK_TO_UNICODE[42028] := 16#F744;
   // GBK_TO_UNICODE[42029] := 16#9C40;
   // GBK_TO_UNICODE[42030] := 16#F745;
   // GBK_TO_UNICODE[42031] := 16#9C41;
   // GBK_TO_UNICODE[42032] := 16#F746;
   // GBK_TO_UNICODE[42033] := 16#9C42;
   // GBK_TO_UNICODE[42034] := 16#F747;
   // GBK_TO_UNICODE[42035] := 16#9C43;
   // GBK_TO_UNICODE[42036] := 16#F748;
   // GBK_TO_UNICODE[42037] := 16#9C44;
   // GBK_TO_UNICODE[42038] := 16#F749;
   // GBK_TO_UNICODE[42039] := 16#9C45;
   // GBK_TO_UNICODE[42040] := 16#F74A;
   // GBK_TO_UNICODE[42041] := 16#9C46;
   // GBK_TO_UNICODE[42042] := 16#F74B;
   // GBK_TO_UNICODE[42043] := 16#9C47;
   // GBK_TO_UNICODE[42044] := 16#F74C;
   // GBK_TO_UNICODE[42045] := 16#9C48;
   // GBK_TO_UNICODE[42046] := 16#F74D;
   // GBK_TO_UNICODE[42047] := 16#9C49;
   // GBK_TO_UNICODE[42048] := 16#F74E;
   // GBK_TO_UNICODE[42049] := 16#9C4A;
   // GBK_TO_UNICODE[42050] := 16#F74F;
   // GBK_TO_UNICODE[42051] := 16#9C4B;
   // GBK_TO_UNICODE[42052] := 16#F750;
   // GBK_TO_UNICODE[42053] := 16#9C4C;
   // GBK_TO_UNICODE[42054] := 16#F751;
   // GBK_TO_UNICODE[42055] := 16#9C4D;
   // GBK_TO_UNICODE[42056] := 16#F752;
   // GBK_TO_UNICODE[42057] := 16#9C4E;
   // GBK_TO_UNICODE[42058] := 16#F753;
   // GBK_TO_UNICODE[42059] := 16#9C4F;
   // GBK_TO_UNICODE[42060] := 16#F754;
   // GBK_TO_UNICODE[42061] := 16#9C50;
   // GBK_TO_UNICODE[42062] := 16#F755;
   // GBK_TO_UNICODE[42063] := 16#9C51;
   // GBK_TO_UNICODE[42064] := 16#F756;
   // GBK_TO_UNICODE[42065] := 16#9C52;
   // GBK_TO_UNICODE[42066] := 16#F757;
   // GBK_TO_UNICODE[42067] := 16#9C53;
